LIN {X 0,Y 412.811,Z 882.496,A -85,B 0,C 180,E1 9709.918,E2 9709.918} C_VEL
LIN {X 0,Y 400.987,Z 919.927,A -85,B 0,C 180,E1 9708.865,E2 9708.865} C_VEL
LIN {X 0,Y 390.445,Z 950.291,A -85,B 0,C 180,E1 9707.777,E2 9707.777} C_VEL
LIN {X 0,Y 381.073,Z 973.005,A -85,B 0,C 180,E1 9706.758,E2 9706.758} C_VEL
LIN {X 0,Y 370.343,Z 995.885,A -85,B 0,C 180,E1 9705.507,E2 9705.507} C_VEL
LIN {X 0,Y 359.142,Z 1016.75,A -85,B 0,C 180,E1 9704.125,E2 9704.125} C_VEL
LIN {X 0,Y 346.722,Z 1037.419,A -85,B 0,C 180,E1 9702.455,E2 9702.455} C_VEL
LIN {X 0,Y 333.977,Z 1056.717,A -85,B 0,C 180,E1 9700.566,E2 9700.566} C_VEL
LIN {X 0,Y 320.046,Z 1075.683,A -85,B 0,C 180,E1 9698.278,E2 9698.278} C_VEL
LIN {X 0,Y 305.349,Z 1094.042,A -85,B 0,C 180,E1 9695.544,E2 9695.544} C_VEL
LIN {X 0,Y 291.757,Z 1109.715,A -85,B 0,C 180,E1 9692.662,E2 9692.662} C_VEL
LIN {X 0,Y 277.905,Z 1124.551,A -85,B 0,C 180,E1 9689.275,E2 9689.275} C_VEL
LIN {X 0,Y 264,Z 1138.62,A -85,B 0,C 180,E1 9685.267,E2 9685.267} C_VEL
LIN {X 0,Y 251.34,Z 1150.739,A -85,B 0,C 180,E1 9680.868,E2 9680.868} C_VEL
LIN {X 0,Y 239.156,Z 1162.034,A -85,B 0,C 180,E1 9675.633,E2 9675.633} C_VEL
LIN {X 0,Y 228.894,Z 1171.576,A -85,B 0,C 180,E1 9669.947,E2 9669.947} C_VEL
LIN {X 0,Y 220.104,Z 1179.984,A -85,B 0,C 180,E1 9663.341,E2 9663.341} C_VEL
LIN {X 0,Y 214.036,Z 1186.297,A -85,B 0,C 180,E1 9656.642,E2 9656.642} C_VEL
LIN {X 0,Y 210.026,Z 1191.417,A -85,B 0,C 180,E1 9649.174,E2 9649.174} C_VEL
LIN {X 0,Y 208.387,Z 1194.571,A -85,B 0,C 180,E1 9642.466,E2 9642.466} C_VEL
LIN {X 0,Y 208.029,Z 1196.144,A -85,B 0,C 180,E1 9636.621,E2 9636.621} C_VEL
LIN {X 0,Y 208.033,Z 1196.749,A -85,B 0,C 180,E1 9631.649,E2 9631.649} C_VEL
LIN {X 0,Y 208.017,Z 1196.626,A -85,B 0,C 180,E1 9626.414,E2 9626.414} C_VEL
LIN {X 0,Y 208.118,Z 1195.498,A -85,B 0,C 180,E1 9620.595,E2 9620.595} C_VEL
LIN {X 0,Y 209.018,Z 1193.143,A -85,B 0,C 180,E1 9614.173,E2 9614.173} C_VEL
LIN {X 0,Y 211.787,Z 1188.974,A -85,B 0,C 180,E1 9606.926,E2 9606.926} C_VEL
LIN {X 0,Y 216.9,Z 1183.182,A -85,B 0,C 180,E1 9599.832,E2 9599.832} C_VEL
LIN {X 0,Y 224.53,Z 1175.655,A -85,B 0,C 180,E1 9593.042,E2 9593.042} C_VEL
LIN {X 0,Y 234.651,Z 1166.193,A -85,B 0,C 180,E1 9586.679,E2 9586.679} C_VEL
LIN {X 0,Y 246.387,Z 1155.288,A -85,B 0,C 180,E1 9581.104,E2 9581.104} C_VEL
LIN {X 0,Y 259.941,Z 1142.471,A -85,B 0,C 180,E1 9576.053,E2 9576.053} C_VEL
LIN {X 0,Y 274.508,Z 1128.008,A -85,B 0,C 180,E1 9571.636,E2 9571.636} C_VEL
LIN {X 0,Y 289.503,Z 1112.12,A -85,B 0,C 180,E1 9567.846,E2 9567.846} C_VEL
LIN {X 0,Y 304.615,Z 1094.805,A -85,B 0,C 180,E1 9564.595,E2 9564.595} C_VEL
LIN {X 0,Y 319.981,Z 1075.607,A -85,B 0,C 180,E1 9561.727,E2 9561.727} C_VEL
LIN {X 0,Y 328.871,Z 1063.516,A -85,B 0,C 180,E1 9560.187,E2 9560.187} C_VEL
LIN {X 0,Y 312.273,Z 1075.955,A -85,B 0,C 180,E1 9558.869,E2 9558.869} C_VEL
LIN {X 0,Y 297.771,Z 1085.65,A -85,B 0,C 180,E1 9557.389,E2 9557.389} C_VEL
LIN {X 0,Y 282.8,Z 1094.747,A -85,B 0,C 180,E1 9555.483,E2 9555.483} C_VEL
LIN {X 0,Y 266.567,Z 1103.684,A -85,B 0,C 180,E1 9552.764,E2 9552.764} C_VEL
LIN {X 0,Y 252.428,Z 1110.885,A -85,B 0,C 180,E1 9549.577,E2 9549.577} C_VEL
LIN {X 0,Y 239.931,Z 1116.966,A -85,B 0,C 180,E1 9545.74,E2 9545.74} C_VEL
LIN {X 0,Y 229.73,Z 1121.893,A -85,B 0,C 180,E1 9541.247,E2 9541.247} C_VEL
LIN {X 0,Y 222.245,Z 1125.755,A -85,B 0,C 180,E1 9536.13,E2 9536.13} C_VEL
LIN {X 0,Y 217.444,Z 1129.147,A -85,B 0,C 180,E1 9529.936,E2 9529.936} C_VEL
LIN {X 0,Y 216.311,Z 1132.47,A -85,B 0,C 180,E1 9522.227,E2 9522.227} C_VEL
LIN {X 0,Y 222.255,Z 1135.612,A -85,B 0,C 180,E1 9512.394,E2 9512.394} C_VEL
LIN {X 0,Y 232.046,Z 1137.189,A -85,B 0,C 180,E1 9505.633,E2 9505.633} C_VEL
LIN {X 0,Y 243.185,Z 1137.819,A -85,B 0,C 180,E1 9500.714,E2 9500.714} C_VEL
LIN {X 0,Y 248.344,Z 1138.002,A -85,B 0,C 180,E1 9498.89,E2 9498.89} C_VEL
LIN {X 0,Y 235.847,Z 1150.144,A -85,B 0,C 180,E1 9493.048,E2 9493.048} C_VEL
LIN {X 0,Y 226.4,Z 1159.496,A -85,B 0,C 180,E1 9487.236,E2 9487.236} C_VEL
LIN {X 0,Y 218.613,Z 1167.518,A -85,B 0,C 180,E1 9480.697,E2 9480.697} C_VEL
LIN {X 0,Y 213.472,Z 1173.506,A -85,B 0,C 180,E1 9474.345,E2 9474.345} C_VEL
LIN {X 0,Y 210.092,Z 1178.183,A -85,B 0,C 180,E1 9467.451,E2 9467.451} C_VEL
LIN {X 0,Y 208.659,Z 1180.906,A -85,B 0,C 180,E1 9461.614,E2 9461.614} C_VEL
LIN {X 0,Y 208.156,Z 1182.441,A -85,B 0,C 180,E1 9456.346,E2 9456.346} C_VEL
LIN {X 0,Y 208.039,Z 1183.097,A -85,B 0,C 180,E1 9451.105,E2 9451.105} C_VEL
LIN {X 0,Y 208.082,Z 1182.855,A -85,B 0,C 180,E1 9445.594,E2 9445.594} C_VEL
LIN {X 0,Y 208.499,Z 1181.364,A -85,B 0,C 180,E1 9439.457,E2 9439.457} C_VEL
LIN {X 0,Y 209.703,Z 1178.846,A -85,B 0,C 180,E1 9433.665,E2 9433.665} C_VEL
LIN {X 0,Y 212.119,Z 1175.235,A -85,B 0,C 180,E1 9427.849,E2 9427.849} C_VEL
LIN {X 0,Y 217.157,Z 1169.21,A -85,B 0,C 180,E1 9420.79,E2 9420.79} C_VEL
LIN {X 0,Y 223.269,Z 1162.652,A -85,B 0,C 180,E1 9415.028,E2 9415.028} C_VEL
LIN {X 0,Y 232.367,Z 1153.659,A -85,B 0,C 180,E1 9408.829,E2 9408.829} C_VEL
LIN {X 0,Y 242.696,Z 1143.563,A -85,B 0,C 180,E1 9403.475,E2 9403.475} C_VEL
LIN {X 0,Y 255.719,Z 1130.948,A -85,B 0,C 180,E1 9398.199,E2 9398.199} C_VEL
LIN {X 0,Y 269.356,Z 1117.324,A -85,B 0,C 180,E1 9393.751,E2 9393.751} C_VEL
LIN {X 0,Y 283.658,Z 1102.296,A -85,B 0,C 180,E1 9389.878,E2 9389.878} C_VEL
LIN {X 0,Y 298.703,Z 1085.671,A -85,B 0,C 180,E1 9386.437,E2 9386.437} C_VEL
LIN {X 0,Y 313.12,Z 1068.459,A -85,B 0,C 180,E1 9383.591,E2 9383.591} C_VEL
LIN {X 0,Y 328.199,Z 1048.906,A -85,B 0,C 180,E1 9380.976,E2 9380.976} C_VEL
LIN {X 0,Y 341.827,Z 1029.717,A -85,B 0,C 180,E1 9378.875,E2 9378.875} C_VEL
LIN {X 0,Y 354.578,Z 1009.676,A -85,B 0,C 180,E1 9377.077,E2 9377.077} C_VEL
LIN {X 0,Y 366.366,Z 989.445,A -85,B 0,C 180,E1 9375.557,E2 9375.557} C_VEL
LIN {X 0,Y 377.497,Z 967.721,A -85,B 0,C 180,E1 9374.213,E2 9374.213} C_VEL
LIN {X 0,Y 388.399,Z 943.457,A -85,B 0,C 180,E1 9372.97,E2 9372.97} C_VEL
LIN {X 0,Y 397.147,Z 920.974,A -85,B 0,C 180,E1 9372.021,E2 9372.021} C_VEL
LIN {X 0,Y 404.369,Z 898.632,A -85,B 0,C 180,E1 9371.242,E2 9371.242} C_VEL
LIN {X 0,Y 414.435,Z 862.441,A -85,B 0,C 180,E1 9370.241,E2 9370.241} C_VEL
LIN {X 0,Y 426.056,Z 818.405,A -85,B 0,C 180,E1 9369.31,E2 9369.31} C_VEL
LIN {X 0,Y 438.723,Z 764.98,A -85,B 0,C 180,E1 9368.335,E2 9368.335} C_VEL
LIN {X 0,Y 449.507,Z 713.302,A -85,B 0,C 180,E1 9367.481,E2 9367.481} C_VEL
LIN {X 0,Y 450.16,Z 709.951,A -85,B 0,C 180,E1 9367.428,E2 9367.428} C_VEL
LIN {X 0,Y 450.433,Z 708.03,A -85,B 0,C 180,E1 9367.262,E2 9367.262} C_VEL
LIN {X 0,Y 450.405,Z 706.776,A -85,B 0,C 180,E1 9366.857,E2 9366.857} C_VEL
LIN {X 0,Y 449.978,Z 706.897,A -85,B 0,C 180,E1 9366.225,E2 9366.225} C_VEL
LIN {X 0,Y 449.184,Z 708.816,A -85,B 0,C 180,E1 9365.494,E2 9365.494} C_VEL
LIN {X 0,Y 447.901,Z 713.065,A -85,B 0,C 180,E1 9364.548,E2 9364.548} C_VEL
LIN {X 0,Y 446.794,Z 717.422,A -85,B 0,C 180,E1 9363.944,E2 9363.944} C_VEL
LIN {X 0,Y 446.052,Z 720.595,A -85,B 0,C 180,E1 9363.669,E2 9363.669} C_VEL
LIN {X 0,Y 439.226,Z 751.426,A -85,B 0,C 180,E1 9361.414,E2 9361.414} C_VEL
LIN {X 0,Y 433.442,Z 778.701,A -85,B 0,C 180,E1 9359.091,E2 9359.091} C_VEL
LIN {X 0,Y 428.161,Z 805.619,A -85,B 0,C 180,E1 9356.469,E2 9356.469} C_VEL
LIN {X 0,Y 423.543,Z 833.332,A -85,B 0,C 180,E1 9353.323,E2 9353.323} C_VEL
LIN {X 0,Y 421.82,Z 845.943,A -85,B 0,C 180,E1 9351.764,E2 9351.764} C_VEL
LIN {X 0,Y 410.531,Z 884.456,A -85,B 0,C 180,E1 9350.964,E2 9350.964} C_VEL
LIN {X 0,Y 399.026,Z 920.276,A -85,B 0,C 180,E1 9349.979,E2 9349.979} C_VEL
LIN {X 0,Y 389.372,Z 947.984,A -85,B 0,C 180,E1 9349.024,E2 9349.024} C_VEL
LIN {X 0,Y 380.15,Z 970.147,A -85,B 0,C 180,E1 9348.071,E2 9348.071} C_VEL
LIN {X 0,Y 370.437,Z 991.045,A -85,B 0,C 180,E1 9346.999,E2 9346.999} C_VEL
LIN {X 0,Y 358.755,Z 1012.769,A -85,B 0,C 180,E1 9345.638,E2 9345.638} C_VEL
LIN {X 0,Y 345.857,Z 1034.272,A -85,B 0,C 180,E1 9343.992,E2 9343.992} C_VEL
LIN {X 0,Y 333.329,Z 1053.021,A -85,B 0,C 180,E1 9342.242,E2 9342.242} C_VEL
LIN {X 0,Y 318.984,Z 1072.455,A -85,B 0,C 180,E1 9340.021,E2 9340.021} C_VEL
LIN {X 0,Y 305.01,Z 1089.89,A -85,B 0,C 180,E1 9337.579,E2 9337.579} C_VEL
LIN {X 0,Y 290.724,Z 1106.062,A -85,B 0,C 180,E1 9334.754,E2 9334.754} C_VEL
LIN {X 0,Y 275.774,Z 1121.883,A -85,B 0,C 180,E1 9331.327,E2 9331.327} C_VEL
LIN {X 0,Y 261.809,Z 1135.683,A -85,B 0,C 180,E1 9327.562,E2 9327.562} C_VEL
LIN {X 0,Y 248.369,Z 1148.138,A -85,B 0,C 180,E1 9323.233,E2 9323.233} C_VEL
LIN {X 0,Y 235.833,Z 1159.442,A -85,B 0,C 180,E1 9318.258,E2 9318.258} C_VEL
LIN {X 0,Y 224.154,Z 1169.717,A -85,B 0,C 180,E1 9312.338,E2 9312.338} C_VEL
LIN {X 0,Y 215.079,Z 1177.78,A -85,B 0,C 180,E1 9306.182,E2 9306.182} C_VEL
LIN {X 0,Y 207.746,Z 1184.836,A -85,B 0,C 180,E1 9299.081,E2 9299.081} C_VEL
LIN {X 0,Y 203.146,Z 1190.016,A -85,B 0,C 180,E1 9291.963,E2 9291.963} C_VEL
LIN {X 0,Y 200.806,Z 1193.468,A -85,B 0,C 180,E1 9284.982,E2 9284.982} C_VEL
LIN {X 0,Y 200.073,Z 1195.622,A -85,B 0,C 180,E1 9278.296,E2 9278.296} C_VEL
LIN {X 0,Y 200.028,Z 1196.434,A -85,B 0,C 180,E1 9272.575,E2 9272.575} C_VEL
LIN {X 0,Y 200.03,Z 1196.45,A -85,B 0,C 180,E1 9267.705,E2 9267.705} C_VEL
LIN {X 0,Y 200.058,Z 1195.716,A -85,B 0,C 180,E1 9262.241,E2 9262.241} C_VEL
LIN {X 0,Y 200.693,Z 1193.696,A -85,B 0,C 180,E1 9255.572,E2 9255.572} C_VEL
LIN {X 0,Y 202.881,Z 1190.321,A -85,B 0,C 180,E1 9248.607,E2 9248.607} C_VEL
LIN {X 0,Y 207.413,Z 1185.146,A -85,B 0,C 180,E1 9241.329,E2 9241.329} C_VEL
LIN {X 0,Y 214.755,Z 1178.072,A -85,B 0,C 180,E1 9234.077,E2 9234.077} C_VEL
LIN {X 0,Y 224.587,Z 1169.279,A -85,B 0,C 180,E1 9227.408,E2 9227.408} C_VEL
LIN {X 0,Y 236.348,Z 1158.936,A -85,B 0,C 180,E1 9221.509,E2 9221.509} C_VEL
LIN {X 0,Y 249.547,Z 1147.037,A -85,B 0,C 180,E1 9216.35,E2 9216.35} C_VEL
LIN {X 0,Y 264.395,Z 1133.053,A -85,B 0,C 180,E1 9211.686,E2 9211.686} C_VEL
LIN {X 0,Y 279.252,Z 1118.218,A -85,B 0,C 180,E1 9207.818,E2 9207.818} C_VEL
LIN {X 0,Y 294.414,Z 1101.886,A -85,B 0,C 180,E1 9204.466,E2 9204.466} C_VEL
LIN {X 0,Y 309.643,Z 1084.032,A -85,B 0,C 180,E1 9201.561,E2 9201.561} C_VEL
LIN {X 0,Y 315.577,Z 1076.646,A -85,B 0,C 180,E1 9200.52,E2 9200.52} C_VEL
LIN {X 0,Y 298.12,Z 1088.173,A -85,B 0,C 180,E1 9198.942,E2 9198.942} C_VEL
LIN {X 0,Y 281.163,Z 1098.148,A -85,B 0,C 180,E1 9196.929,E2 9196.929} C_VEL
LIN {X 0,Y 264.092,Z 1107.202,A -85,B 0,C 180,E1 9194.238,E2 9194.238} C_VEL
LIN {X 0,Y 250.119,Z 1113.928,A -85,B 0,C 180,E1 9191.296,E2 9191.296} C_VEL
LIN {X 0,Y 237.074,Z 1119.968,A -85,B 0,C 180,E1 9187.617,E2 9187.617} C_VEL
LIN {X 0,Y 227.218,Z 1124.381,A -85,B 0,C 180,E1 9183.785,E2 9183.785} C_VEL
LIN {X 0,Y 218.049,Z 1128.64,A -85,B 0,C 180,E1 9178.613,E2 9178.613} C_VEL
LIN {X 0,Y 211.262,Z 1132.587,A -85,B 0,C 180,E1 9171.563,E2 9171.563} C_VEL
LIN {X 0,Y 209.204,Z 1136.12,A -85,B 0,C 180,E1 9162.763,E2 9162.763} C_VEL
LIN {X 0,Y 215.054,Z 1139.294,A -85,B 0,C 180,E1 9152.293,E2 9152.293} C_VEL
LIN {X 0,Y 225.258,Z 1140.856,A -85,B 0,C 180,E1 9145.067,E2 9145.067} C_VEL
LIN {X 0,Y 237.163,Z 1141.564,A -85,B 0,C 180,E1 9139.83,E2 9139.83} C_VEL
LIN {X 0,Y 239.46,Z 1141.692,A -85,B 0,C 180,E1 9138.933,E2 9138.933} C_VEL
LIN {X 0,Y 228.015,Z 1152.144,A -85,B 0,C 180,E1 9133.513,E2 9133.513} C_VEL
LIN {X 0,Y 218.012,Z 1161.542,A -85,B 0,C 180,E1 9127.261,E2 9127.261} C_VEL
LIN {X 0,Y 210.559,Z 1168.836,A -85,B 0,C 180,E1 9120.858,E2 9120.858} C_VEL
LIN {X 0,Y 204.789,Z 1175.208,A -85,B 0,C 180,E1 9113.376,E2 9113.376} C_VEL
LIN {X 0,Y 201.976,Z 1178.973,A -85,B 0,C 180,E1 9107.164,E2 9107.164} C_VEL
LIN {X 0,Y 200.563,Z 1181.603,A -85,B 0,C 180,E1 9100.924,E2 9100.924} C_VEL
LIN {X 0,Y 200.092,Z 1183.11,A -85,B 0,C 180,E1 9094.589,E2 9094.589} C_VEL
LIN {X 0,Y 200.043,Z 1183.37,A -85,B 0,C 180,E1 9088.858,E2 9088.858} C_VEL
LIN {X 0,Y 200.17,Z 1182.736,A -85,B 0,C 180,E1 9083.406,E2 9083.406} C_VEL
LIN {X 0,Y 200.718,Z 1181.223,A -85,B 0,C 180,E1 9077.927,E2 9077.927} C_VEL
LIN {X 0,Y 202.181,Z 1178.677,A -85,B 0,C 180,E1 9072.148,E2 9072.148} C_VEL
LIN {X 0,Y 205.577,Z 1174.375,A -85,B 0,C 180,E1 9065.278,E2 9065.278} C_VEL
LIN {X 0,Y 211.111,Z 1168.293,A -85,B 0,C 180,E1 9058.489,E2 9058.489} C_VEL
LIN {X 0,Y 218.999,Z 1160.714,A -85,B 0,C 180,E1 9051.953,E2 9051.953} C_VEL
LIN {X 0,Y 228.792,Z 1151.499,A -85,B 0,C 180,E1 9045.988,E2 9045.988} C_VEL
LIN {X 0,Y 240.607,Z 1140.727,A -85,B 0,C 180,E1 9040.498,E2 9040.498} C_VEL
LIN {X 0,Y 254.213,Z 1127.965,A -85,B 0,C 180,E1 9035.499,E2 9035.499} C_VEL
LIN {X 0,Y 269.411,Z 1113.153,A -85,B 0,C 180,E1 9030.988,E2 9030.988} C_VEL
LIN {X 0,Y 284.568,Z 1097.649,A -85,B 0,C 180,E1 9027.263,E2 9027.263} C_VEL
LIN {X 0,Y 300.298,Z 1080.229,A -85,B 0,C 180,E1 9023.968,E2 9023.968} C_VEL
LIN {X 0,Y 316.161,Z 1061.208,A -85,B 0,C 180,E1 9021.106,E2 9021.106} C_VEL
LIN {X 0,Y 330.628,Z 1042.445,A -85,B 0,C 180,E1 9018.822,E2 9018.822} C_VEL
LIN {X 0,Y 344.691,Z 1022.113,A -85,B 0,C 180,E1 9016.819,E2 9016.819} C_VEL
LIN {X 0,Y 358.519,Z 999.958,A -85,B 0,C 180,E1 9015.033,E2 9015.033} C_VEL
LIN {X 0,Y 370.366,Z 978.771,A -85,B 0,C 180,E1 9013.625,E2 9013.625} C_VEL
LIN {X 0,Y 380.429,Z 958.054,A -85,B 0,C 180,E1 9012.479,E2 9012.479} C_VEL
LIN {X 0,Y 389.747,Z 936.743,A -85,B 0,C 180,E1 9011.487,E2 9011.487} C_VEL
LIN {X 0,Y 397.779,Z 914.776,A -85,B 0,C 180,E1 9010.641,E2 9010.641} C_VEL
LIN {X 0,Y 404.743,Z 893.101,A -85,B 0,C 180,E1 9009.944,E2 9009.944} C_VEL
LIN {X 0,Y 416.476,Z 850.737,A -85,B 0,C 180,E1 9008.867,E2 9008.867} C_VEL
LIN {X 0,Y 429.491,Z 800.675,A -85,B 0,C 180,E1 9007.911,E2 9007.911} C_VEL
LIN {X 0,Y 441.609,Z 748.272,A -85,B 0,C 180,E1 9007.011,E2 9007.011} C_VEL
LIN {X 0,Y 452.336,Z 694.609,A -85,B 0,C 180,E1 9006.178,E2 9006.178} C_VEL
LIN {X 0,Y 452.794,Z 692.087,A -85,B 0,C 180,E1 9006.121,E2 9006.121} C_VEL
LIN {X 0,Y 452.304,Z 692.999,A -85,B 0,C 180,E1 9005.574,E2 9005.574} C_VEL
LIN {X 0,Y 446.052,Z 720.595,A -85,B 0,C 180,E1 9003.669,E2 9003.669} C_VEL
LIN {X 0,Y 444.49,Z 727.708,A -85,B 0,C 180,E1 9003.32,E2 9003.32} C_VEL
LIN {X 0,Y 440.022,Z 747.992,A -85,B 0,C 180,E1 9002.766,E2 9002.766} C_VEL
LIN {X 0,Y 438.677,Z 753.942,A -85,B 0,C 180,E1 9002.427,E2 9002.427} C_VEL
LIN {X 0,Y 432.402,Z 781.506,A -85,B 0,C 180,E1 9000.099,E2 9000.099} C_VEL
LIN {X 0,Y 426.937,Z 806.918,A -85,B 0,C 180,E1 8997.651,E2 8997.651} C_VEL
LIN {X 0,Y 421.776,Z 834.64,A -85,B 0,C 180,E1 8994.559,E2 8994.559} C_VEL
LIN {X 0,Y 419.509,Z 849.049,A -85,B 0,C 180,E1 8992.782,E2 8992.782} C_VEL
LIN {X 0,Y 407.591,Z 888.947,A -85,B 0,C 180,E1 8991.962,E2 8991.962} C_VEL
LIN {X 0,Y 395.608,Z 925.572,A -85,B 0,C 180,E1 8990.955,E2 8990.955} C_VEL
LIN {X 0,Y 386.691,Z 950.05,A -85,B 0,C 180,E1 8990.106,E2 8990.106} C_VEL
LIN {X 0,Y 378.853,Z 968.601,A -85,B 0,C 180,E1 8989.329,E2 8989.329} C_VEL
LIN {X 0,Y 369.103,Z 989.382,A -85,B 0,C 180,E1 8988.306,E2 8988.306} C_VEL
LIN {X 0,Y 358.011,Z 1009.79,A -85,B 0,C 180,E1 8987.077,E2 8987.077} C_VEL
LIN {X 0,Y 346.237,Z 1029.583,A -85,B 0,C 180,E1 8985.657,E2 8985.657} C_VEL
LIN {X 0,Y 332.966,Z 1049.316,A -85,B 0,C 180,E1 8983.925,E2 8983.925} C_VEL
LIN {X 0,Y 317.96,Z 1069.51,A -85,B 0,C 180,E1 8981.74,E2 8981.74} C_VEL
LIN {X 0,Y 304.238,Z 1086.387,A -85,B 0,C 180,E1 8979.489,E2 8979.489} C_VEL
LIN {X 0,Y 288.712,Z 1103.847,A -85,B 0,C 180,E1 8976.594,E2 8976.594} C_VEL
LIN {X 0,Y 273.228,Z 1119.915,A -85,B 0,C 180,E1 8973.236,E2 8973.236} C_VEL
LIN {X 0,Y 259.02,Z 1133.559,A -85,B 0,C 180,E1 8969.622,E2 8969.622} C_VEL
LIN {X 0,Y 244.002,Z 1147.15,A -85,B 0,C 180,E1 8965.036,E2 8965.036} C_VEL
LIN {X 0,Y 230.815,Z 1158.549,A -85,B 0,C 180,E1 8960.058,E2 8960.058} C_VEL
LIN {X 0,Y 218.904,Z 1168.528,A -85,B 0,C 180,E1 8954.33,E2 8954.33} C_VEL
LIN {X 0,Y 208.625,Z 1177.205,A -85,B 0,C 180,E1 8947.739,E2 8947.739} C_VEL
LIN {X 0,Y 200.7,Z 1184.31,A -85,B 0,C 180,E1 8940.47,E2 8940.47} C_VEL
LIN {X 0,Y 195.6,Z 1189.596,A -85,B 0,C 180,E1 8933.052,E2 8933.052} C_VEL
LIN {X 0,Y 192.933,Z 1193.182,A -85,B 0,C 180,E1 8925.63,E2 8925.63} C_VEL
LIN {X 0,Y 192.08,Z 1195.378,A -85,B 0,C 180,E1 8918.48,E2 8918.48} C_VEL
LIN {X 0,Y 192.032,Z 1196.169,A -85,B 0,C 180,E1 8912.682,E2 8912.682} C_VEL
LIN {X 0,Y 192.033,Z 1196.186,A -85,B 0,C 180,E1 8907.609,E2 8907.609} C_VEL
LIN {X 0,Y 192.069,Z 1195.445,A -85,B 0,C 180,E1 8901.916,E2 8901.916} C_VEL
LIN {X 0,Y 192.801,Z 1193.412,A -85,B 0,C 180,E1 8894.968,E2 8894.968} C_VEL
LIN {X 0,Y 195.221,Z 1190.016,A -85,B 0,C 180,E1 8887.724,E2 8887.724} C_VEL
LIN {X 0,Y 200.259,Z 1184.711,A -85,B 0,C 180,E1 8880.043,E2 8880.043} C_VEL
LIN {X 0,Y 208.374,Z 1177.393,A -85,B 0,C 180,E1 8872.449,E2 8872.449} C_VEL
LIN {X 0,Y 218.914,Z 1168.479,A -85,B 0,C 180,E1 8865.663,E2 8865.663} C_VEL
LIN {X 0,Y 231.361,Z 1158.036,A -85,B 0,C 180,E1 8859.707,E2 8859.707} C_VEL
LIN {X 0,Y 245.377,Z 1145.87,A -85,B 0,C 180,E1 8854.501,E2 8854.501} C_VEL
LIN {X 0,Y 260.73,Z 1131.884,A -85,B 0,C 180,E1 8849.904,E2 8849.904} C_VEL
LIN {X 0,Y 276.89,Z 1116.111,A -85,B 0,C 180,E1 8845.91,E2 8845.91} C_VEL
LIN {X 0,Y 292.537,Z 1099.608,A -85,B 0,C 180,E1 8842.648,E2 8842.648} C_VEL
LIN {X 0,Y 302.365,Z 1088.426,A -85,B 0,C 180,E1 8840.806,E2 8840.806} C_VEL
LIN {X 0,Y 284.426,Z 1098.878,A -85,B 0,C 180,E1 8838.97,E2 8838.97} C_VEL
LIN {X 0,Y 267.69,Z 1107.72,A -85,B 0,C 180,E1 8836.715,E2 8836.715} C_VEL
LIN {X 0,Y 252.346,Z 1115.038,A -85,B 0,C 180,E1 8833.987,E2 8833.987} C_VEL
LIN {X 0,Y 238.031,Z 1121.349,A -85,B 0,C 180,E1 8830.582,E2 8830.582} C_VEL
LIN {X 0,Y 225.412,Z 1126.726,A -85,B 0,C 180,E1 8826.453,E2 8826.453} C_VEL
LIN {X 0,Y 215.059,Z 1131.104,A -85,B 0,C 180,E1 8821.504,E2 8821.504} C_VEL
LIN {X 0,Y 207.526,Z 1134.572,A -85,B 0,C 180,E1 8815.855,E2 8815.855} C_VEL
LIN {X 0,Y 202.41,Z 1138.234,A -85,B 0,C 180,E1 8807.446,E2 8807.446} C_VEL
LIN {X 0,Y 203.621,Z 1141.241,A -85,B 0,C 180,E1 8798.087,E2 8798.087} C_VEL
LIN {X 0,Y 210.765,Z 1143.45,A -85,B 0,C 180,E1 8789.495,E2 8789.495} C_VEL
LIN {X 0,Y 222.632,Z 1144.699,A -85,B 0,C 180,E1 8782.352,E2 8782.352} C_VEL
LIN {X 0,Y 230.538,Z 1145.066,A -85,B 0,C 180,E1 8779.001,E2 8779.001} C_VEL
LIN {X 0,Y 218.868,Z 1155.373,A -85,B 0,C 180,E1 8773.26,E2 8773.26} C_VEL
LIN {X 0,Y 208.902,Z 1164.124,A -85,B 0,C 180,E1 8766.752,E2 8766.752} C_VEL
LIN {X 0,Y 201.1,Z 1171.519,A -85,B 0,C 180,E1 8759.491,E2 8759.491} C_VEL
LIN {X 0,Y 196.371,Z 1176.499,A -85,B 0,C 180,E1 8752.77,E2 8752.77} C_VEL
LIN {X 0,Y 193.569,Z 1180.224,A -85,B 0,C 180,E1 8745.892,E2 8745.892} C_VEL
LIN {X 0,Y 192.354,Z 1182.536,A -85,B 0,C 180,E1 8738.975,E2 8738.975} C_VEL
LIN {X 0,Y 192.066,Z 1183.477,A -85,B 0,C 180,E1 8733.286,E2 8733.286} C_VEL
LIN {X 0,Y 192.05,Z 1183.589,A -85,B 0,C 180,E1 8728.214,E2 8728.214} C_VEL
LIN {X 0,Y 192.206,Z 1182.937,A -85,B 0,C 180,E1 8722.832,E2 8722.832} C_VEL
LIN {X 0,Y 192.852,Z 1181.391,A -85,B 0,C 180,E1 8717.122,E2 8717.122} C_VEL
LIN {X 0,Y 194.65,Z 1178.667,A -85,B 0,C 180,E1 8710.811,E2 8710.811} C_VEL
LIN {X 0,Y 198.945,Z 1173.722,A -85,B 0,C 180,E1 8703.111,E2 8703.111} C_VEL
LIN {X 0,Y 204.582,Z 1168.146,A -85,B 0,C 180,E1 8696.816,E2 8696.816} C_VEL
LIN {X 0,Y 213.277,Z 1160.304,A -85,B 0,C 180,E1 8690.043,E2 8690.043} C_VEL
LIN {X 0,Y 223.85,Z 1151.036,A -85,B 0,C 180,E1 8684.021,E2 8684.021} C_VEL
LIN {X 0,Y 237.519,Z 1139.058,A -85,B 0,C 180,E1 8678.08,E2 8678.08} C_VEL
LIN {X 0,Y 252.012,Z 1126.11,A -85,B 0,C 180,E1 8673.164,E2 8673.164} C_VEL
LIN {X 0,Y 267.301,Z 1111.6,A -85,B 0,C 180,E1 8668.924,E2 8668.924} C_VEL
LIN {X 0,Y 283.809,Z 1094.958,A -85,B 0,C 180,E1 8665.125,E2 8665.125} C_VEL
LIN {X 0,Y 299.806,Z 1077.677,A -85,B 0,C 180,E1 8662.012,E2 8662.012} C_VEL
LIN {X 0,Y 314.919,Z 1059.732,A -85,B 0,C 180,E1 8659.448,E2 8659.448} C_VEL
LIN {X 0,Y 330.581,Z 1039.479,A -85,B 0,C 180,E1 8657.111,E2 8657.111} C_VEL
LIN {X 0,Y 344.997,Z 1018.928,A -85,B 0,C 180,E1 8655.189,E2 8655.189} C_VEL
LIN {X 0,Y 357.103,Z 999.454,A -85,B 0,C 180,E1 8653.7,E2 8653.7} C_VEL
LIN {X 0,Y 368.546,Z 979.309,A -85,B 0,C 180,E1 8652.404,E2 8652.404} C_VEL
LIN {X 0,Y 378.32,Z 959.508,A -85,B 0,C 180,E1 8651.335,E2 8651.335} C_VEL
LIN {X 0,Y 387.728,Z 938.49,A -85,B 0,C 180,E1 8650.375,E2 8650.375} C_VEL
LIN {X 0,Y 395.921,Z 916.579,A -85,B 0,C 180,E1 8649.546,E2 8649.546} C_VEL
LIN {X 0,Y 403.228,Z 894.205,A -85,B 0,C 180,E1 8648.841,E2 8648.841} C_VEL
LIN {X 0,Y 415.5,Z 850.931,A -85,B 0,C 180,E1 8647.769,E2 8647.769} C_VEL
LIN {X 0,Y 429.41,Z 798.024,A -85,B 0,C 180,E1 8646.796,E2 8646.796} C_VEL
LIN {X 0,Y 442.417,Z 741.668,A -85,B 0,C 180,E1 8645.867,E2 8645.867} C_VEL
LIN {X 0,Y 448.433,Z 712.167,A -85,B 0,C 180,E1 8645.401,E2 8645.401} C_VEL
LIN {X 0,Y 439.649,Z 749.613,A -85,B 0,C 180,E1 8642.754,E2 8642.754} C_VEL
LIN {X 0,Y 438.677,Z 753.942,A -85,B 0,C 180,E1 8642.427,E2 8642.427} C_VEL
LIN {X 0,Y 437.092,Z 760.897,A -85,B 0,C 180,E1 8642.026,E2 8642.026} C_VEL
LIN {X 0,Y 432.325,Z 780.783,A -85,B 0,C 180,E1 8641.3,E2 8641.3} C_VEL
LIN {X 0,Y 430.941,Z 786.563,A -85,B 0,C 180,E1 8640.91,E2 8640.91} C_VEL
LIN {X 0,Y 425.125,Z 812.174,A -85,B 0,C 180,E1 8638.435,E2 8638.435} C_VEL
LIN {X 0,Y 419.318,Z 841.092,A -85,B 0,C 180,E1 8635.178,E2 8635.178} C_VEL
LIN {X 0,Y 417.366,Z 852.094,A -85,B 0,C 180,E1 8633.813,E2 8633.813} C_VEL
LIN {X 0,Y 405.206,Z 892.313,A -85,B 0,C 180,E1 8633.002,E2 8633.002} C_VEL
LIN {X 0,Y 392.778,Z 929.723,A -85,B 0,C 180,E1 8631.982,E2 8631.982} C_VEL
LIN {X 0,Y 384.439,Z 951.566,A -85,B 0,C 180,E1 8631.226,E2 8631.226} C_VEL
LIN {X 0,Y 374.842,Z 973.68,A -85,B 0,C 180,E1 8630.307,E2 8630.307} C_VEL
LIN {X 0,Y 364.785,Z 993.544,A -85,B 0,C 180,E1 8629.3,E2 8629.3} C_VEL
LIN {X 0,Y 353.562,Z 1013.799,A -85,B 0,C 180,E1 8628.085,E2 8628.085} C_VEL
LIN {X 0,Y 340.805,Z 1033.918,A -85,B 0,C 180,E1 8626.598,E2 8626.598} C_VEL
LIN {X 0,Y 327.732,Z 1052.851,A -85,B 0,C 180,E1 8624.921,E2 8624.921} C_VEL
LIN {X 0,Y 312.912,Z 1071.98,A -85,B 0,C 180,E1 8622.82,E2 8622.82} C_VEL
LIN {X 0,Y 297.337,Z 1090.303,A -85,B 0,C 180,E1 8620.311,E2 8620.311} C_VEL
LIN {X 0,Y 282.353,Z 1106.507,A -85,B 0,C 180,E1 8617.55,E2 8617.55} C_VEL
LIN {X 0,Y 266.576,Z 1122.14,A -85,B 0,C 180,E1 8614.177,E2 8614.177} C_VEL
LIN {X 0,Y 251.062,Z 1136.44,A -85,B 0,C 180,E1 8610.245,E2 8610.245} C_VEL
LIN {X 0,Y 237.359,Z 1148.247,A -85,B 0,C 180,E1 8606.079,E2 8606.079} C_VEL
LIN {X 0,Y 223.251,Z 1159.861,A -85,B 0,C 180,E1 8600.783,E2 8600.783} C_VEL
LIN {X 0,Y 211.06,Z 1169.665,A -85,B 0,C 180,E1 8594.895,E2 8594.895} C_VEL
LIN {X 0,Y 200.659,Z 1177.991,A -85,B 0,C 180,E1 8588.157,E2 8588.157} C_VEL
LIN {X 0,Y 192.811,Z 1184.627,A -85,B 0,C 180,E1 8580.886,E2 8580.886} C_VEL
LIN {X 0,Y 187.596,Z 1189.728,A -85,B 0,C 180,E1 8573.225,E2 8573.225} C_VEL
LIN {X 0,Y 184.949,Z 1193.1,A -85,B 0,C 180,E1 8565.777,E2 8565.777} C_VEL
LIN {X 0,Y 184.082,Z 1195.18,A -85,B 0,C 180,E1 8558.429,E2 8558.429} C_VEL
LIN {X 0,Y 184.035,Z 1195.906,A -85,B 0,C 180,E1 8552.799,E2 8552.799} C_VEL
LIN {X 0,Y 184.039,Z 1195.939,A -85,B 0,C 180,E1 8547.817,E2 8547.817} C_VEL
LIN {X 0,Y 184.065,Z 1195.279,A -85,B 0,C 180,E1 8542.191,E2 8542.191} C_VEL
LIN {X 0,Y 184.729,Z 1193.492,A -85,B 0,C 180,E1 8535.258,E2 8535.258} C_VEL
LIN {X 0,Y 187.151,Z 1190.191,A -85,B 0,C 180,E1 8527.704,E2 8527.704} C_VEL
LIN {X 0,Y 192.364,Z 1185.017,A -85,B 0,C 180,E1 8519.639,E2 8519.639} C_VEL
LIN {X 0,Y 200.423,Z 1178.158,A -85,B 0,C 180,E1 8512.022,E2 8512.022} C_VEL
LIN {X 0,Y 211.069,Z 1169.606,A -85,B 0,C 180,E1 8505.098,E2 8505.098} C_VEL
LIN {X 0,Y 223.808,Z 1159.349,A -85,B 0,C 180,E1 8498.976,E2 8498.976} C_VEL
LIN {X 0,Y 238.625,Z 1147.12,A -85,B 0,C 180,E1 8493.5,E2 8493.5} C_VEL
LIN {X 0,Y 254.497,Z 1133.28,A -85,B 0,C 180,E1 8488.815,E2 8488.815} C_VEL
LIN {X 0,Y 270.995,Z 1117.809,A -85,B 0,C 180,E1 8484.811,E2 8484.811} C_VEL
LIN {X 0,Y 287.018,Z 1101.46,A -85,B 0,C 180,E1 8481.537,E2 8481.537} C_VEL
LIN {X 0,Y 289.307,Z 1098.949,A -85,B 0,C 180,E1 8481.062,E2 8481.062} C_VEL
LIN {X 0,Y 271.912,Z 1108.059,A -85,B 0,C 180,E1 8479.076,E2 8479.076} C_VEL
LIN {X 0,Y 254.352,Z 1116.406,A -85,B 0,C 180,E1 8476.417,E2 8476.417} C_VEL
LIN {X 0,Y 238.16,Z 1123.312,A -85,B 0,C 180,E1 8473.078,E2 8473.078} C_VEL
LIN {X 0,Y 223.699,Z 1129.125,A -85,B 0,C 180,E1 8468.935,E2 8468.935} C_VEL
LIN {X 0,Y 211.883,Z 1133.733,A -85,B 0,C 180,E1 8464.059,E2 8464.059} C_VEL
LIN {X 0,Y 202.893,Z 1137.441,A -85,B 0,C 180,E1 8458.306,E2 8458.306} C_VEL
LIN {X 0,Y 196.877,Z 1140.612,A -85,B 0,C 180,E1 8451.236,E2 8451.236} C_VEL
LIN {X 0,Y 195.049,Z 1143.6,A -85,B 0,C 180,E1 8442.395,E2 8442.395} C_VEL
LIN {X 0,Y 201.304,Z 1146.465,A -85,B 0,C 180,E1 8431.196,E2 8431.196} C_VEL
LIN {X 0,Y 212.531,Z 1147.861,A -85,B 0,C 180,E1 8423.309,E2 8423.309} C_VEL
LIN {X 0,Y 221.655,Z 1148.402,A -85,B 0,C 180,E1 8419.101,E2 8419.101} C_VEL
LIN {X 0,Y 210.122,Z 1157.898,A -85,B 0,C 180,E1 8413.258,E2 8413.258} C_VEL
LIN {X 0,Y 201.204,Z 1165.4,A -85,B 0,C 180,E1 8407.325,E2 8407.325} C_VEL
LIN {X 0,Y 193.155,Z 1172.526,A -85,B 0,C 180,E1 8399.803,E2 8399.803} C_VEL
LIN {X 0,Y 188.482,Z 1177.17,A -85,B 0,C 180,E1 8393.118,E2 8393.118} C_VEL
LIN {X 0,Y 185.403,Z 1180.995,A -85,B 0,C 180,E1 8385.327,E2 8385.327} C_VEL
LIN {X 0,Y 184.333,Z 1182.927,A -85,B 0,C 180,E1 8378.74,E2 8378.74} C_VEL
LIN {X 0,Y 184.067,Z 1183.76,A -85,B 0,C 180,E1 8373.118,E2 8373.118} C_VEL
LIN {X 0,Y 184.054,Z 1183.854,A -85,B 0,C 180,E1 8368.136,E2 8368.136} C_VEL
LIN {X 0,Y 184.229,Z 1183.205,A -85,B 0,C 180,E1 8362.519,E2 8362.519} C_VEL
LIN {X 0,Y 184.953,Z 1181.663,A -85,B 0,C 180,E1 8356.562,E2 8356.562} C_VEL
LIN {X 0,Y 186.947,Z 1178.946,A -85,B 0,C 180,E1 8349.987,E2 8349.987} C_VEL
LIN {X 0,Y 191.623,Z 1174.011,A -85,B 0,C 180,E1 8341.995,E2 8341.995} C_VEL
LIN {X 0,Y 197.701,Z 1168.467,A -85,B 0,C 180,E1 8335.502,E2 8335.502} C_VEL
LIN {X 0,Y 207.387,Z 1160.276,A -85,B 0,C 180,E1 8328.296,E2 8328.296} C_VEL
LIN {X 0,Y 218.646,Z 1150.99,A -85,B 0,C 180,E1 8322.203,E2 8322.203} C_VEL
LIN {X 0,Y 232.794,Z 1139.167,A -85,B 0,C 180,E1 8316.352,E2 8316.352} C_VEL
LIN {X 0,Y 247.557,Z 1126.51,A -85,B 0,C 180,E1 8311.551,E2 8311.551} C_VEL
LIN {X 0,Y 263.388,Z 1112.031,A -85,B 0,C 180,E1 8307.344,E2 8307.344} C_VEL
LIN {X 0,Y 279.636,Z 1096.183,A -85,B 0,C 180,E1 8303.749,E2 8303.749} C_VEL
LIN {X 0,Y 296.022,Z 1079.061,A -85,B 0,C 180,E1 8300.678,E2 8300.678} C_VEL
LIN {X 0,Y 311.608,Z 1061.086,A -85,B 0,C 180,E1 8298.135,E2 8298.135} C_VEL
LIN {X 0,Y 327.42,Z 1041.16,A -85,B 0,C 180,E1 8295.865,E2 8295.865} C_VEL
LIN {X 0,Y 341.392,Z 1021.784,A -85,B 0,C 180,E1 8294.069,E2 8294.069} C_VEL
LIN {X 0,Y 353.502,Z 1002.924,A -85,B 0,C 180,E1 8292.633,E2 8292.633} C_VEL
LIN {X 0,Y 364.196,Z 984.701,A -85,B 0,C 180,E1 8291.454,E2 8291.454} C_VEL
LIN {X 0,Y 375.006,Z 963.873,A -85,B 0,C 180,E1 8290.318,E2 8290.318} C_VEL
LIN {X 0,Y 383.785,Z 944.873,A -85,B 0,C 180,E1 8289.447,E2 8289.447} C_VEL
LIN {X 0,Y 392.828,Z 922.225,A -85,B 0,C 180,E1 8288.573,E2 8288.573} C_VEL
LIN {X 0,Y 399.923,Z 901.452,A -85,B 0,C 180,E1 8287.904,E2 8287.904} C_VEL
LIN {X 0,Y 411.996,Z 860.655,A -85,B 0,C 180,E1 8286.868,E2 8286.868} C_VEL
LIN {X 0,Y 426.144,Z 808.526,A -85,B 0,C 180,E1 8285.902,E2 8285.902} C_VEL
LIN {X 0,Y 438.788,Z 755.89,A -85,B 0,C 180,E1 8285.044,E2 8285.044} C_VEL
LIN {X 0,Y 442.588,Z 738.476,A -85,B 0,C 180,E1 8284.762,E2 8284.762} C_VEL
LIN {X 0,Y 435.441,Z 767.749,A -85,B 0,C 180,E1 8282.533,E2 8282.533} C_VEL
LIN {X 0,Y 430.941,Z 786.563,A -85,B 0,C 180,E1 8280.91,E2 8280.91} C_VEL
LIN {X 0,Y 429.349,Z 793.362,A -85,B 0,C 180,E1 8280.452,E2 8280.452} C_VEL
LIN {X 0,Y 424.718,Z 811.92,A -85,B 0,C 180,E1 8279.623,E2 8279.623} C_VEL
LIN {X 0,Y 423.084,Z 818.472,A -85,B 0,C 180,E1 8279.114,E2 8279.114} C_VEL
LIN {X 0,Y 417.01,Z 846.356,A -85,B 0,C 180,E1 8275.944,E2 8275.944} C_VEL
LIN {X 0,Y 415.317,Z 855.237,A -85,B 0,C 180,E1 8274.852,E2 8274.852} C_VEL
LIN {X 0,Y 403.575,Z 893.556,A -85,B 0,C 180,E1 8274.099,E2 8274.099} C_VEL
LIN {X 0,Y 391.286,Z 930.132,A -85,B 0,C 180,E1 8273.133,E2 8273.133} C_VEL
LIN {X 0,Y 382.338,Z 953.222,A -85,B 0,C 180,E1 8272.355,E2 8272.355} C_VEL
LIN {X 0,Y 372.098,Z 975.729,A -85,B 0,C 180,E1 8271.428,E2 8271.428} C_VEL
LIN {X 0,Y 361.505,Z 996.346,A -85,B 0,C 180,E1 8270.4,E2 8270.4} C_VEL
LIN {X 0,Y 349.886,Z 1016.222,A -85,B 0,C 180,E1 8269.201,E2 8269.201} C_VEL
LIN {X 0,Y 339.337,Z 1032.592,A -85,B 0,C 180,E1 8268.02,E2 8268.02} C_VEL
LIN {X 0,Y 326.517,Z 1050.967,A -85,B 0,C 180,E1 8266.464,E2 8266.464} C_VEL
LIN {X 0,Y 312.222,Z 1069.167,A -85,B 0,C 180,E1 8264.557,E2 8264.557} C_VEL
LIN {X 0,Y 297.069,Z 1086.994,A -85,B 0,C 180,E1 8262.266,E2 8262.266} C_VEL
LIN {X 0,Y 281.602,Z 1103.446,A -85,B 0,C 180,E1 8259.608,E2 8259.608} C_VEL
LIN {X 0,Y 265.246,Z 1119.449,A -85,B 0,C 180,E1 8256.344,E2 8256.344} C_VEL
LIN {X 0,Y 249.79,Z 1133.506,A -85,B 0,C 180,E1 8252.696,E2 8252.696} C_VEL
LIN {X 0,Y 234.493,Z 1146.334,A -85,B 0,C 180,E1 8248.367,E2 8248.367} C_VEL
LIN {X 0,Y 219.744,Z 1158.089,A -85,B 0,C 180,E1 8243.204,E2 8243.204} C_VEL
LIN {X 0,Y 206.672,Z 1168.146,A -85,B 0,C 180,E1 8237.334,E2 8237.334} C_VEL
LIN {X 0,Y 195.319,Z 1176.692,A -85,B 0,C 180,E1 8230.547,E2 8230.547} C_VEL
LIN {X 0,Y 185.989,Z 1184.063,A -85,B 0,C 180,E1 8222.516,E2 8222.516} C_VEL
LIN {X 0,Y 180.127,Z 1189.331,A -85,B 0,C 180,E1 8214.443,E2 8214.443} C_VEL
LIN {X 0,Y 177.153,Z 1192.734,A -85,B 0,C 180,E1 8206.725,E2 8206.725} C_VEL
LIN {X 0,Y 176.1,Z 1194.895,A -85,B 0,C 180,E1 8198.896,E2 8198.896} C_VEL
LIN {X 0,Y 176.037,Z 1195.641,A -85,B 0,C 180,E1 8192.926,E2 8192.926} C_VEL
LIN {X 0,Y 176.042,Z 1195.676,A -85,B 0,C 180,E1 8187.717,E2 8187.717} C_VEL
LIN {X 0,Y 176.076,Z 1195.013,A -85,B 0,C 180,E1 8181.834,E2 8181.834} C_VEL
LIN {X 0,Y 176.921,Z 1193.091,A -85,B 0,C 180,E1 8174.256,E2 8174.256} C_VEL
LIN {X 0,Y 179.7,Z 1189.721,A -85,B 0,C 180,E1 8166.379,E2 8166.379} C_VEL
LIN {X 0,Y 185.43,Z 1184.505,A -85,B 0,C 180,E1 8158.096,E2 8158.096} C_VEL
LIN {X 0,Y 194.137,Z 1177.599,A -85,B 0,C 180,E1 8150.305,E2 8150.305} C_VEL
LIN {X 0,Y 205.683,Z 1168.841,A -85,B 0,C 180,E1 8143.177,E2 8143.177} C_VEL
LIN {X 0,Y 219.168,Z 1158.48,A -85,B 0,C 180,E1 8137.019,E2 8137.019} C_VEL
LIN {X 0,Y 234.708,Z 1146.101,A -85,B 0,C 180,E1 8131.563,E2 8131.563} C_VEL
LIN {X 0,Y 250.83,Z 1132.452,A -85,B 0,C 180,E1 8127.029,E2 8127.029} C_VEL
LIN {X 0,Y 266.778,Z 1117.932,A -85,B 0,C 180,E1 8123.322,E2 8123.322} C_VEL
LIN {X 0,Y 276.565,Z 1108.372,A -85,B 0,C 180,E1 8121.306,E2 8121.306} C_VEL
LIN {X 0,Y 258.357,Z 1116.937,A -85,B 0,C 180,E1 8118.971,E2 8118.971} C_VEL
LIN {X 0,Y 242.518,Z 1123.699,A -85,B 0,C 180,E1 8116.282,E2 8116.282} C_VEL
LIN {X 0,Y 226.246,Z 1130.01,A -85,B 0,C 180,E1 8112.507,E2 8112.507} C_VEL
LIN {X 0,Y 212.763,Z 1135.014,A -85,B 0,C 180,E1 8108.105,E2 8108.105} C_VEL
LIN {X 0,Y 201.179,Z 1139.251,A -85,B 0,C 180,E1 8102.505,E2 8102.505} C_VEL
LIN {X 0,Y 192.038,Z 1142.987,A -85,B 0,C 180,E1 8094.922,E2 8094.922} C_VEL
LIN {X 0,Y 187.842,Z 1146.158,A -85,B 0,C 180,E1 8085.512,E2 8085.512} C_VEL
LIN {X 0,Y 190.633,Z 1148.835,A -85,B 0,C 180,E1 8075.156,E2 8075.156} C_VEL
LIN {X 0,Y 200.456,Z 1150.729,A -85,B 0,C 180,E1 8065.691,E2 8065.691} C_VEL
LIN {X 0,Y 212.715,Z 1151.566,A -85,B 0,C 180,E1 8059.187,E2 8059.187} C_VEL
LIN {X 0,Y 201.356,Z 1160.422,A -85,B 0,C 180,E1 8053.261,E2 8053.261} C_VEL
LIN {X 0,Y 191.006,Z 1168.648,A -85,B 0,C 180,E1 8045.899,E2 8045.899} C_VEL
LIN {X 0,Y 184.44,Z 1174.209,A -85,B 0,C 180,E1 8039.207,E2 8039.207} C_VEL
LIN {X 0,Y 179.323,Z 1179.174,A -85,B 0,C 180,E1 8030.911,E2 8030.911} C_VEL
LIN {X 0,Y 177.091,Z 1181.896,A -85,B 0,C 180,E1 8024.055,E2 8024.055} C_VEL
LIN {X 0,Y 176.264,Z 1183.446,A -85,B 0,C 180,E1 8017.829,E2 8017.829} C_VEL
LIN {X 0,Y 176.059,Z 1184.108,A -85,B 0,C 180,E1 8011.957,E2 8011.957} C_VEL
LIN {X 0,Y 176.079,Z 1184.012,A -85,B 0,C 180,E1 8006.423,E2 8006.423} C_VEL
LIN {X 0,Y 176.435,Z 1183.099,A -85,B 0,C 180,E1 8000.215,E2 8000.215} C_VEL
LIN {X 0,Y 178.042,Z 1180.69,A -85,B 0,C 180,E1 7992.351,E2 7992.351} C_VEL
LIN {X 0,Y 181.282,Z 1177.159,A -85,B 0,C 180,E1 7985.221,E2 7985.221} C_VEL
LIN {X 0,Y 186.821,Z 1172.237,A -85,B 0,C 180,E1 7978.009,E2 7978.009} C_VEL
LIN {X 0,Y 195.744,Z 1164.92,A -85,B 0,C 180,E1 7970.324,E2 7970.324} C_VEL
LIN {X 0,Y 206.927,Z 1156.237,A -85,B 0,C 180,E1 7963.553,E2 7963.553} C_VEL
LIN {X 0,Y 220.423,Z 1145.589,A -85,B 0,C 180,E1 7957.46,E2 7957.46} C_VEL
LIN {X 0,Y 236.282,Z 1132.746,A -85,B 0,C 180,E1 7951.936,E2 7951.936} C_VEL
LIN {X 0,Y 252.419,Z 1119.048,A -85,B 0,C 180,E1 7947.47,E2 7947.47} C_VEL
LIN {X 0,Y 267.933,Z 1104.784,A -85,B 0,C 180,E1 7943.901,E2 7943.901} C_VEL
LIN {X 0,Y 283.536,Z 1089.619,A -85,B 0,C 180,E1 7940.858,E2 7940.858} C_VEL
LIN {X 0,Y 298.983,Z 1073.198,A -85,B 0,C 180,E1 7938.245,E2 7938.245} C_VEL
LIN {X 0,Y 315.288,Z 1054.285,A -85,B 0,C 180,E1 7935.827,E2 7935.827} C_VEL
LIN {X 0,Y 328.279,Z 1037.753,A -85,B 0,C 180,E1 7934.103,E2 7934.103} C_VEL
LIN {X 0,Y 342.425,Z 1017.94,A -85,B 0,C 180,E1 7932.393,E2 7932.393} C_VEL
LIN {X 0,Y 354.52,Z 999.225,A -85,B 0,C 180,E1 7931.053,E2 7931.053} C_VEL
LIN {X 0,Y 366.321,Z 978.576,A -85,B 0,C 180,E1 7929.831,E2 7929.831} C_VEL
LIN {X 0,Y 376.095,Z 959.554,A -85,B 0,C 180,E1 7928.87,E2 7928.87} C_VEL
LIN {X 0,Y 386.127,Z 937.015,A -85,B 0,C 180,E1 7927.924,E2 7927.924} C_VEL
LIN {X 0,Y 394.985,Z 913.959,A -85,B 0,C 180,E1 7927.121,E2 7927.121} C_VEL
LIN {X 0,Y 405.584,Z 880.158,A -85,B 0,C 180,E1 7926.191,E2 7926.191} C_VEL
LIN {X 0,Y 417.821,Z 837.614,A -85,B 0,C 180,E1 7925.309,E2 7925.309} C_VEL
LIN {X 0,Y 430.758,Z 788.266,A -85,B 0,C 180,E1 7924.495,E2 7924.495} C_VEL
LIN {X 0,Y 436.685,Z 763.616,A -85,B 0,C 180,E1 7924.099,E2 7924.099} C_VEL
LIN {X 0,Y 429.521,Z 791.933,A -85,B 0,C 180,E1 7921.701,E2 7921.701} C_VEL
LIN {X 0,Y 423.084,Z 818.472,A -85,B 0,C 180,E1 7919.114,E2 7919.114} C_VEL
LIN {X 0,Y 421.513,Z 825.009,A -85,B 0,C 180,E1 7918.583,E2 7918.583} C_VEL
LIN {X 0,Y 416.852,Z 843.111,A -85,B 0,C 180,E1 7917.571,E2 7917.571} C_VEL
LIN {X 0,Y 415.345,Z 849.423,A -85,B 0,C 180,E1 7916.993,E2 7916.993} C_VEL
LIN {X 0,Y 413.492,Z 858.122,A -85,B 0,C 180,E1 7915.905,E2 7915.905} C_VEL
LIN {X 0,Y 400.889,Z 898.411,A -85,B 0,C 180,E1 7915.124,E2 7915.124} C_VEL
LIN {X 0,Y 389.461,Z 931.856,A -85,B 0,C 180,E1 7914.253,E2 7914.253} C_VEL
LIN {X 0,Y 380.386,Z 954.776,A -85,B 0,C 180,E1 7913.499,E2 7913.499} C_VEL
LIN {X 0,Y 369.549,Z 977.907,A -85,B 0,C 180,E1 7912.564,E2 7912.564} C_VEL
LIN {X 0,Y 356.965,Z 1001.263,A -85,B 0,C 180,E1 7911.391,E2 7911.391} C_VEL
LIN {X 0,Y 344.986,Z 1020.998,A -85,B 0,C 180,E1 7910.193,E2 7910.193} C_VEL
LIN {X 0,Y 331.185,Z 1041.183,A -85,B 0,C 180,E1 7908.683,E2 7908.683} C_VEL
LIN {X 0,Y 319.761,Z 1056.449,A -85,B 0,C 180,E1 7907.309,E2 7907.309} C_VEL
LIN {X 0,Y 305.284,Z 1074.294,A -85,B 0,C 180,E1 7905.392,E2 7905.392} C_VEL
LIN {X 0,Y 290.379,Z 1090.811,A -85,B 0,C 180,E1 7903.177,E2 7903.177} C_VEL
LIN {X 0,Y 273.886,Z 1107.684,A -85,B 0,C 180,E1 7900.362,E2 7900.362} C_VEL
LIN {X 0,Y 257.93,Z 1122.57,A -85,B 0,C 180,E1 7897.191,E2 7897.191} C_VEL
LIN {X 0,Y 241.631,Z 1136.578,A -85,B 0,C 180,E1 7893.35,E2 7893.35} C_VEL
LIN {X 0,Y 226.324,Z 1148.946,A -85,B 0,C 180,E1 7888.983,E2 7888.983} C_VEL
LIN {X 0,Y 211.157,Z 1160.321,A -85,B 0,C 180,E1 7883.603,E2 7883.603} C_VEL
LIN {X 0,Y 197.42,Z 1170.288,A -85,B 0,C 180,E1 7877.25,E2 7877.25} C_VEL
LIN {X 0,Y 186.11,Z 1178.477,A -85,B 0,C 180,E1 7870.138,E2 7870.138} C_VEL
LIN {X 0,Y 177.504,Z 1184.922,A -85,B 0,C 180,E1 7862.332,E2 7862.332} C_VEL
LIN {X 0,Y 171.747,Z 1189.812,A -85,B 0,C 180,E1 7853.93,E2 7853.93} C_VEL
LIN {X 0,Y 168.838,Z 1193.163,A -85,B 0,C 180,E1 7845.451,E2 7845.451} C_VEL
LIN {X 0,Y 168.079,Z 1194.799,A -85,B 0,C 180,E1 7838.204,E2 7838.204} C_VEL
LIN {X 0,Y 168.045,Z 1195.414,A -85,B 0,C 180,E1 7832.383,E2 7832.383} C_VEL
LIN {X 0,Y 168.038,Z 1195.376,A -85,B 0,C 180,E1 7826.926,E2 7826.926} C_VEL
LIN {X 0,Y 168.115,Z 1194.632,A -85,B 0,C 180,E1 7820.755,E2 7820.755} C_VEL
LIN {X 0,Y 169.243,Z 1192.56,A -85,B 0,C 180,E1 7812.814,E2 7812.814} C_VEL
LIN {X 0,Y 172.531,Z 1189.096,A -85,B 0,C 180,E1 7804.601,E2 7804.601} C_VEL
LIN {X 0,Y 179.021,Z 1183.709,A -85,B 0,C 180,E1 7796.041,E2 7796.041} C_VEL
LIN {X 0,Y 189.036,Z 1176.275,A -85,B 0,C 180,E1 7787.776,E2 7787.776} C_VEL
LIN {X 0,Y 201.05,Z 1167.675,A -85,B 0,C 180,E1 7780.888,E2 7780.888} C_VEL
LIN {X 0,Y 215.415,Z 1157.122,A -85,B 0,C 180,E1 7774.753,E2 7774.753} C_VEL
LIN {X 0,Y 231.059,Z 1145.057,A -85,B 0,C 180,E1 7769.559,E2 7769.559} C_VEL
LIN {X 0,Y 248.236,Z 1130.942,A -85,B 0,C 180,E1 7764.997,E2 7764.997} C_VEL
LIN {X 0,Y 263.966,Z 1116.935,A -85,B 0,C 180,E1 7761.528,E2 7761.528} C_VEL
LIN {X 0,Y 245.978,Z 1124.596,A -85,B 0,C 180,E1 7758.978,E2 7758.978} C_VEL
LIN {X 0,Y 229.045,Z 1131.046,A -85,B 0,C 180,E1 7755.704,E2 7755.704} C_VEL
LIN {X 0,Y 213.045,Z 1136.678,A -85,B 0,C 180,E1 7751.369,E2 7751.369} C_VEL
LIN {X 0,Y 200.174,Z 1141.044,A -85,B 0,C 180,E1 7746.309,E2 7746.309} C_VEL
LIN {X 0,Y 189.989,Z 1144.548,A -85,B 0,C 180,E1 7740.138,E2 7740.138} C_VEL
LIN {X 0,Y 182.83,Z 1147.663,A -85,B 0,C 180,E1 7732.142,E2 7732.142} C_VEL
LIN {X 0,Y 180.563,Z 1150.391,A -85,B 0,C 180,E1 7722.6,E2 7722.6} C_VEL
LIN {X 0,Y 187.117,Z 1153.056,A -85,B 0,C 180,E1 7710.201,E2 7710.201} C_VEL
LIN {X 0,Y 199.332,Z 1154.296,A -85,B 0,C 180,E1 7701.537,E2 7701.537} C_VEL
LIN {X 0,Y 203.796,Z 1154.589,A -85,B 0,C 180,E1 7699.295,E2 7699.295} C_VEL
LIN {X 0,Y 190.817,Z 1164.143,A -85,B 0,C 180,E1 7692.127,E2 7692.127} C_VEL
LIN {X 0,Y 181.872,Z 1170.879,A -85,B 0,C 180,E1 7685.262,E2 7685.262} C_VEL
LIN {X 0,Y 174.555,Z 1176.795,A -85,B 0,C 180,E1 7676.91,E2 7676.91} C_VEL
LIN {X 0,Y 170.815,Z 1180.321,A -85,B 0,C 180,E1 7669.851,E2 7669.851} C_VEL
LIN {X 0,Y 168.72,Z 1182.992,A -85,B 0,C 180,E1 7661.975,E2 7661.975} C_VEL
LIN {X 0,Y 168.114,Z 1184.21,A -85,B 0,C 180,E1 7654.781,E2 7654.781} C_VEL
LIN {X 0,Y 168.061,Z 1184.421,A -85,B 0,C 180,E1 7648.641,E2 7648.641} C_VEL
LIN {X 0,Y 168.24,Z 1183.859,A -85,B 0,C 180,E1 7642.491,E2 7642.491} C_VEL
LIN {X 0,Y 169.072,Z 1182.398,A -85,B 0,C 180,E1 7635.907,E2 7635.907} C_VEL
LIN {X 0,Y 171.199,Z 1179.955,A -85,B 0,C 180,E1 7629.133,E2 7629.133} C_VEL
LIN {X 0,Y 176.172,Z 1175.534,A -85,B 0,C 180,E1 7620.789,E2 7620.789} C_VEL
LIN {X 0,Y 183.533,Z 1169.652,A -85,B 0,C 180,E1 7613.187,E2 7613.187} C_VEL
LIN {X 0,Y 194.119,Z 1161.819,A -85,B 0,C 180,E1 7605.724,E2 7605.724} C_VEL
LIN {X 0,Y 206.682,Z 1152.526,A -85,B 0,C 180,E1 7599.288,E2 7599.288} C_VEL
LIN {X 0,Y 222.345,Z 1140.7,A -85,B 0,C 180,E1 7593.24,E2 7593.24} C_VEL
LIN {X 0,Y 237.858,Z 1128.498,A -85,B 0,C 180,E1 7588.536,E2 7588.536} C_VEL
LIN {X 0,Y 253.916,Z 1114.859,A -85,B 0,C 180,E1 7584.552,E2 7584.552} C_VEL
LIN {X 0,Y 270.208,Z 1100.201,A -85,B 0,C 180,E1 7581.18,E2 7581.18} C_VEL
LIN {X 0,Y 285.622,Z 1085.087,A -85,B 0,C 180,E1 7578.442,E2 7578.442} C_VEL
LIN {X 0,Y 302.88,Z 1066.68,A -85,B 0,C 180,E1 7575.79,E2 7575.79} C_VEL
LIN {X 0,Y 318.501,Z 1048.457,A -85,B 0,C 180,E1 7573.693,E2 7573.693} C_VEL
LIN {X 0,Y 332.235,Z 1030.468,A -85,B 0,C 180,E1 7572.023,E2 7572.023} C_VEL
LIN {X 0,Y 344.423,Z 1013.261,A -85,B 0,C 180,E1 7570.673,E2 7570.673} C_VEL
LIN {X 0,Y 357.219,Z 992.871,A -85,B 0,C 180,E1 7569.343,E2 7569.343} C_VEL
LIN {X 0,Y 369.208,Z 971.621,A -85,B 0,C 180,E1 7568.191,E2 7568.191} C_VEL
LIN {X 0,Y 379.938,Z 949.482,A -85,B 0,C 180,E1 7567.203,E2 7567.203} C_VEL
LIN {X 0,Y 390.03,Z 925.278,A -85,B 0,C 180,E1 7566.31,E2 7566.31} C_VEL
LIN {X 0,Y 398.289,Z 901.807,A -85,B 0,C 180,E1 7565.6,E2 7565.6} C_VEL
LIN {X 0,Y 410.933,Z 860.146,A -85,B 0,C 180,E1 7564.618,E2 7564.618} C_VEL
LIN {X 0,Y 424.001,Z 813.56,A -85,B 0,C 180,E1 7563.819,E2 7563.819} C_VEL
LIN {X 0,Y 430.813,Z 787.165,A -85,B 0,C 180,E1 7563.402,E2 7563.402} C_VEL
LIN {X 0,Y 423.902,Z 813.641,A -85,B 0,C 180,E1 7560.929,E2 7560.929} C_VEL
LIN {X 0,Y 418.546,Z 835.306,A -85,B 0,C 180,E1 7558.631,E2 7558.631} C_VEL
LIN {X 0,Y 415.345,Z 849.423,A -85,B 0,C 180,E1 7556.993,E2 7556.993} C_VEL
LIN {X 0,Y 414.5,Z 853.045,A -85,B 0,C 180,E1 7556.679,E2 7556.679} C_VEL
LIN {X 0,Y 412.719,Z 859.248,A -85,B 0,C 180,E1 7556.465,E2 7556.465} C_VEL
LIN {X 0,Y 409.99,Z 867.954,A -85,B 0,C 180,E1 7556.481,E2 7556.481} C_VEL
LIN {X 0,Y 405.875,Z 880.33,A -85,B 0,C 180,E1 7556.609,E2 7556.609} C_VEL
LIN {X 0,Y 404.829,Z 883.706,A -85,B 0,C 180,E1 7556.572,E2 7556.572} C_VEL
LIN {X 0,Y 392.043,Z 922.239,A -85,B 0,C 180,E1 7555.698,E2 7555.698} C_VEL
LIN {X 0,Y 383.374,Z 944.762,A -85,B 0,C 180,E1 7555.042,E2 7555.042} C_VEL
LIN {X 0,Y 373.808,Z 966.639,A -85,B 0,C 180,E1 7554.271,E2 7554.271} C_VEL
LIN {X 0,Y 362.412,Z 988.842,A -85,B 0,C 180,E1 7553.307,E2 7553.307} C_VEL
LIN {X 0,Y 349.259,Z 1011.499,A -85,B 0,C 180,E1 7552.1,E2 7552.1} C_VEL
LIN {X 0,Y 336.57,Z 1030.816,A -85,B 0,C 180,E1 7550.842,E2 7550.842} C_VEL
LIN {X 0,Y 321.63,Z 1051.167,A -85,B 0,C 180,E1 7549.214,E2 7549.214} C_VEL
LIN {X 0,Y 309.051,Z 1066.747,A -85,B 0,C 180,E1 7547.694,E2 7547.694} C_VEL
LIN {X 0,Y 293.63,Z 1084.339,A -85,B 0,C 180,E1 7545.606,E2 7545.606} C_VEL
LIN {X 0,Y 278.684,Z 1099.705,A -85,B 0,C 180,E1 7543.318,E2 7543.318} C_VEL
LIN {X 0,Y 262.953,Z 1114.77,A -85,B 0,C 180,E1 7540.556,E2 7540.556} C_VEL
LIN {X 0,Y 246.303,Z 1129.23,A -85,B 0,C 180,E1 7537.141,E2 7537.141} C_VEL
LIN {X 0,Y 229.126,Z 1143.012,A -85,B 0,C 180,E1 7532.895,E2 7532.895} C_VEL
LIN {X 0,Y 213.136,Z 1155.054,A -85,B 0,C 180,E1 7527.986,E2 7527.986} C_VEL
LIN {X 0,Y 197.88,Z 1165.74,A -85,B 0,C 180,E1 7522.017,E2 7522.017} C_VEL
LIN {X 0,Y 184.743,Z 1174.692,A -85,B 0,C 180,E1 7515.149,E2 7515.149} C_VEL
LIN {X 0,Y 174.24,Z 1181.971,A -85,B 0,C 180,E1 7507.46,E2 7507.46} C_VEL
LIN {X 0,Y 166.431,Z 1187.713,A -85,B 0,C 180,E1 7498.721,E2 7498.721} C_VEL
LIN {X 0,Y 161.982,Z 1191.661,A -85,B 0,C 180,E1 7489.842,E2 7489.842} C_VEL
LIN {X 0,Y 160.277,Z 1194.021,A -85,B 0,C 180,E1 7481.636,E2 7481.636} C_VEL
LIN {X 0,Y 160.033,Z 1195.038,A -85,B 0,C 180,E1 7474.654,E2 7474.654} C_VEL
LIN {X 0,Y 160.059,Z 1195.219,A -85,B 0,C 180,E1 7468.922,E2 7468.922} C_VEL
LIN {X 0,Y 160.067,Z 1194.687,A -85,B 0,C 180,E1 7462.458,E2 7462.458} C_VEL
LIN {X 0,Y 160.695,Z 1193.235,A -85,B 0,C 180,E1 7455.215,E2 7455.215} C_VEL
LIN {X 0,Y 163.576,Z 1190.094,A -85,B 0,C 180,E1 7446.202,E2 7446.202} C_VEL
LIN {X 0,Y 169.335,Z 1185.477,A -85,B 0,C 180,E1 7437.493,E2 7437.493} C_VEL
LIN {X 0,Y 178.519,Z 1178.919,A -85,B 0,C 180,E1 7429.052,E2 7429.052} C_VEL
LIN {X 0,Y 191.164,Z 1170.297,A -85,B 0,C 180,E1 7421.227,E2 7421.227} C_VEL
LIN {X 0,Y 205.96,Z 1160.039,A -85,B 0,C 180,E1 7414.612,E2 7414.612} C_VEL
LIN {X 0,Y 222.085,Z 1148.365,A -85,B 0,C 180,E1 7409.134,E2 7409.134} C_VEL
LIN {X 0,Y 238.704,Z 1135.376,A -85,B 0,C 180,E1 7404.631,E2 7404.631} C_VEL
LIN {X 0,Y 251.33,Z 1124.821,A -85,B 0,C 180,E1 7401.715,E2 7401.715} C_VEL
LIN {X 0,Y 233.862,Z 1131.507,A -85,B 0,C 180,E1 7398.962,E2 7398.962} C_VEL
LIN {X 0,Y 216.552,Z 1137.461,A -85,B 0,C 180,E1 7395.19,E2 7395.19} C_VEL
LIN {X 0,Y 201.626,Z 1142.272,A -85,B 0,C 180,E1 7390.573,E2 7390.573} C_VEL
LIN {X 0,Y 188.577,Z 1146.331,A -85,B 0,C 180,E1 7384.529,E2 7384.529} C_VEL
LIN {X 0,Y 178.138,Z 1149.889,A -85,B 0,C 180,E1 7376.138,E2 7376.138} C_VEL
LIN {X 0,Y 173.32,Z 1152.86,A -85,B 0,C 180,E1 7365.637,E2 7365.637} C_VEL
LIN {X 0,Y 176.378,Z 1155.309,A -85,B 0,C 180,E1 7354.118,E2 7354.118} C_VEL
LIN {X 0,Y 186.507,Z 1156.908,A -85,B 0,C 180,E1 7344.242,E2 7344.242} C_VEL
LIN {X 0,Y 194.842,Z 1157.525,A -85,B 0,C 180,E1 7339.425,E2 7339.425} C_VEL
LIN {X 0,Y 182.462,Z 1166.063,A -85,B 0,C 180,E1 7332.384,E2 7332.384} C_VEL
LIN {X 0,Y 171.903,Z 1173.567,A -85,B 0,C 180,E1 7323.718,E2 7323.718} C_VEL
LIN {X 0,Y 165.84,Z 1178.237,A -85,B 0,C 180,E1 7316.056,E2 7316.056} C_VEL
LIN {X 0,Y 161.877,Z 1181.928,A -85,B 0,C 180,E1 7307.251,E2 7307.251} C_VEL
LIN {X 0,Y 160.438,Z 1183.791,A -85,B 0,C 180,E1 7299.692,E2 7299.692} C_VEL
LIN {X 0,Y 160.088,Z 1184.552,A -85,B 0,C 180,E1 7293.585,E2 7293.585} C_VEL
LIN {X 0,Y 160.069,Z 1184.643,A -85,B 0,C 180,E1 7287.856,E2 7287.856} C_VEL
LIN {X 0,Y 160.295,Z 1184.067,A -85,B 0,C 180,E1 7281.756,E2 7281.756} C_VEL
LIN {X 0,Y 161.28,Z 1182.592,A -85,B 0,C 180,E1 7274.912,E2 7274.912} C_VEL
LIN {X 0,Y 163.905,Z 1179.953,A -85,B 0,C 180,E1 7267.403,E2 7267.403} C_VEL
LIN {X 0,Y 169.857,Z 1175.14,A -85,B 0,C 180,E1 7258.41,E2 7258.41} C_VEL
LIN {X 0,Y 177.806,Z 1169.373,A -85,B 0,C 180,E1 7250.9,E2 7250.9} C_VEL
LIN {X 0,Y 189.992,Z 1160.916,A -85,B 0,C 180,E1 7242.992,E2 7242.992} C_VEL
LIN {X 0,Y 203.893,Z 1151.267,A -85,B 0,C 180,E1 7236.469,E2 7236.469} C_VEL
LIN {X 0,Y 219.225,Z 1140.072,A -85,B 0,C 180,E1 7230.974,E2 7230.974} C_VEL
LIN {X 0,Y 235.457,Z 1127.71,A -85,B 0,C 180,E1 7226.367,E2 7226.367} C_VEL
LIN {X 0,Y 252.148,Z 1114.031,A -85,B 0,C 180,E1 7222.498,E2 7222.498} C_VEL
LIN {X 0,Y 269.788,Z 1098.361,A -85,B 0,C 180,E1 7219.087,E2 7219.087} C_VEL
LIN {X 0,Y 286.532,Z 1082.31,A -85,B 0,C 180,E1 7216.344,E2 7216.344} C_VEL
LIN {X 0,Y 301.26,Z 1066.606,A -85,B 0,C 180,E1 7214.218,E2 7214.218} C_VEL
LIN {X 0,Y 316.668,Z 1049.025,A -85,B 0,C 180,E1 7212.258,E2 7212.258} C_VEL
LIN {X 0,Y 332.003,Z 1029.298,A -85,B 0,C 180,E1 7210.497,E2 7210.497} C_VEL
LIN {X 0,Y 346.811,Z 1008.088,A -85,B 0,C 180,E1 7208.957,E2 7208.957} C_VEL
LIN {X 0,Y 359.238,Z 988.19,A -85,B 0,C 180,E1 7207.766,E2 7207.766} C_VEL
LIN {X 0,Y 370.969,Z 966.616,A -85,B 0,C 180,E1 7206.693,E2 7206.693} C_VEL
LIN {X 0,Y 381.39,Z 944.895,A -85,B 0,C 180,E1 7205.797,E2 7205.797} C_VEL
LIN {X 0,Y 389.965,Z 923.784,A -85,B 0,C 180,E1 7205.071,E2 7205.071} C_VEL
LIN {X 0,Y 398.114,Z 900.522,A -85,B 0,C 180,E1 7204.406,E2 7204.406} C_VEL
LIN {X 0,Y 410.422,Z 860.631,A -85,B 0,C 180,E1 7203.504,E2 7203.504} C_VEL
LIN {X 0,Y 422.872,Z 817.117,A -85,B 0,C 180,E1 7202.787,E2 7202.787} C_VEL
LIN {X 0,Y 424.89,Z 809.584,A -85,B 0,C 180,E1 7202.652,E2 7202.652} C_VEL
LIN {X 0,Y 417.777,Z 836.426,A -85,B 0,C 180,E1 7199.897,E2 7199.897} C_VEL
LIN {X 0,Y 411.868,Z 860.519,A -85,B 0,C 180,E1 7197.043,E2 7197.043} C_VEL
LIN {X 0,Y 411.517,Z 861.865,A -85,B 0,C 180,E1 7196.954,E2 7196.954} C_VEL
LIN {X 0,Y 404.829,Z 883.706,A -85,B 0,C 180,E1 7196.572,E2 7196.572} C_VEL
LIN {X 0,Y 402.421,Z 891.093,A -85,B 0,C 180,E1 7196.567,E2 7196.567} C_VEL
LIN {X 0,Y 395.232,Z 910.797,A -85,B 0,C 180,E1 7197.038,E2 7197.038} C_VEL
LIN {X 0,Y 393.068,Z 917.075,A -85,B 0,C 180,E1 7197.001,E2 7197.001} C_VEL
LIN {X 0,Y 384.695,Z 939.343,A -85,B 0,C 180,E1 7196.407,E2 7196.407} C_VEL
LIN {X 0,Y 376.937,Z 957.356,A -85,B 0,C 180,E1 7195.832,E2 7195.832} C_VEL
LIN {X 0,Y 366.938,Z 978.199,A -85,B 0,C 180,E1 7195.048,E2 7195.048} C_VEL
LIN {X 0,Y 354.856,Z 999.784,A -85,B 0,C 180,E1 7194.048,E2 7194.048} C_VEL
LIN {X 0,Y 341.598,Z 1021.051,A -85,B 0,C 180,E1 7192.854,E2 7192.854} C_VEL
LIN {X 0,Y 327.105,Z 1041.496,A -85,B 0,C 180,E1 7191.423,E2 7191.423} C_VEL
LIN {X 0,Y 310.719,Z 1062.156,A -85,B 0,C 180,E1 7189.618,E2 7189.618} C_VEL
LIN {X 0,Y 297.276,Z 1077.545,A -85,B 0,C 180,E1 7187.963,E2 7187.963} C_VEL
LIN {X 0,Y 280.703,Z 1094.898,A -85,B 0,C 180,E1 7185.657,E2 7185.657} C_VEL
LIN {X 0,Y 266.116,Z 1108.758,A -85,B 0,C 180,E1 7183.348,E2 7183.348} C_VEL
LIN {X 0,Y 249.556,Z 1123.429,A -85,B 0,C 180,E1 7180.306,E2 7180.306} C_VEL
LIN {X 0,Y 232.201,Z 1137.389,A -85,B 0,C 180,E1 7176.511,E2 7176.511} C_VEL
LIN {X 0,Y 215.208,Z 1149.97,A -85,B 0,C 180,E1 7171.97,E2 7171.97} C_VEL
LIN {X 0,Y 199.641,Z 1160.843,A -85,B 0,C 180,E1 7166.755,E2 7166.755} C_VEL
LIN {X 0,Y 184.716,Z 1170.603,A -85,B 0,C 180,E1 7160.227,E2 7160.227} C_VEL
LIN {X 0,Y 171.818,Z 1178.868,A -85,B 0,C 180,E1 7152.452,E2 7152.452} C_VEL
LIN {X 0,Y 162.358,Z 1185.186,A -85,B 0,C 180,E1 7144.08,E2 7144.08} C_VEL
LIN {X 0,Y 156.237,Z 1189.655,A -85,B 0,C 180,E1 7135.385,E2 7135.385} C_VEL
LIN {X 0,Y 152.898,Z 1192.87,A -85,B 0,C 180,E1 7125.937,E2 7125.937} C_VEL
LIN {X 0,Y 152.087,Z 1194.37,A -85,B 0,C 180,E1 7118.312,E2 7118.312} C_VEL
LIN {X 0,Y 152.058,Z 1194.927,A -85,B 0,C 180,E1 7111.789,E2 7111.789} C_VEL
LIN {X 0,Y 152.038,Z 1194.81,A -85,B 0,C 180,E1 7105.847,E2 7105.847} C_VEL
LIN {X 0,Y 152.251,Z 1193.921,A -85,B 0,C 180,E1 7098.633,E2 7098.633} C_VEL
LIN {X 0,Y 154.019,Z 1191.616,A -85,B 0,C 180,E1 7089.87,E2 7089.87} C_VEL
LIN {X 0,Y 158.886,Z 1187.62,A -85,B 0,C 180,E1 7080.28,E2 7080.28} C_VEL
LIN {X 0,Y 166.907,Z 1182.076,A -85,B 0,C 180,E1 7071.457,E2 7071.457} C_VEL
LIN {X 0,Y 178.413,Z 1174.605,A -85,B 0,C 180,E1 7063.229,E2 7063.229} C_VEL
LIN {X 0,Y 192.811,Z 1165.264,A -85,B 0,C 180,E1 7055.997,E2 7055.997} C_VEL
LIN {X 0,Y 208.94,Z 1154.392,A -85,B 0,C 180,E1 7049.977,E2 7049.977} C_VEL
LIN {X 0,Y 226.152,Z 1141.881,A -85,B 0,C 180,E1 7044.986,E2 7044.986} C_VEL
LIN {X 0,Y 238.822,Z 1132.041,A -85,B 0,C 180,E1 7041.878,E2 7041.878} C_VEL
LIN {X 0,Y 220.545,Z 1138.271,A -85,B 0,C 180,E1 7038.632,E2 7038.632} C_VEL
LIN {X 0,Y 203.14,Z 1143.653,A -85,B 0,C 180,E1 7034.247,E2 7034.247} C_VEL
LIN {X 0,Y 188.556,Z 1147.896,A -85,B 0,C 180,E1 7028.846,E2 7028.846} C_VEL
LIN {X 0,Y 177.107,Z 1151.199,A -85,B 0,C 180,E1 7022.265,E2 7022.265} C_VEL
LIN {X 0,Y 168.785,Z 1154.121,A -85,B 0,C 180,E1 7013.537,E2 7013.537} C_VEL
LIN {X 0,Y 165.855,Z 1156.675,A -85,B 0,C 180,E1 7002.818,E2 7002.818} C_VEL
LIN {X 0,Y 172.476,Z 1159.036,A -85,B 0,C 180,E1 6989.325,E2 6989.325} C_VEL
LIN {X 0,Y 185.656,Z 1160.159,A -85,B 0,C 180,E1 6979.738,E2 6979.738} C_VEL
LIN {X 0,Y 185.767,Z 1160.271,A -85,B 0,C 180,E1 6979.521,E2 6979.521} C_VEL
LIN {X 0,Y 173.208,Z 1168.545,A -85,B 0,C 180,E1 6972.044,E2 6972.044} C_VEL
LIN {X 0,Y 163.562,Z 1174.913,A -85,B 0,C 180,E1 6963.757,E2 6963.757} C_VEL
LIN {X 0,Y 156.801,Z 1179.885,A -85,B 0,C 180,E1 6954.492,E2 6954.492} C_VEL
LIN {X 0,Y 153.567,Z 1182.711,A -85,B 0,C 180,E1 6946.263,E2 6946.263} C_VEL
LIN {X 0,Y 152.375,Z 1184.24,A -85,B 0,C 180,E1 6939.066,E2 6939.066} C_VEL
LIN {X 0,Y 152.077,Z 1184.875,A -85,B 0,C 180,E1 6932.643,E2 6932.643} C_VEL
LIN {X 0,Y 152.081,Z 1184.866,A -85,B 0,C 180,E1 6926.99,E2 6926.99} C_VEL
LIN {X 0,Y 152.403,Z 1184.213,A -85,B 0,C 180,E1 6920.564,E2 6920.564} C_VEL
LIN {X 0,Y 153.647,Z 1182.662,A -85,B 0,C 180,E1 6913.366,E2 6913.366} C_VEL
LIN {X 0,Y 157.369,Z 1179.511,A -85,B 0,C 180,E1 6904.407,E2 6904.407} C_VEL
LIN {X 0,Y 164.187,Z 1174.53,A -85,B 0,C 180,E1 6895.509,E2 6895.509} C_VEL
LIN {X 0,Y 174.003,Z 1168.078,A -85,B 0,C 180,E1 6887.313,E2 6887.313} C_VEL
LIN {X 0,Y 186.584,Z 1159.818,A -85,B 0,C 180,E1 6879.982,E2 6879.982} C_VEL
LIN {X 0,Y 202.513,Z 1149.202,A -85,B 0,C 180,E1 6873.234,E2 6873.234} C_VEL
LIN {X 0,Y 218.604,Z 1138.013,A -85,B 0,C 180,E1 6868.029,E2 6868.029} C_VEL
LIN {X 0,Y 235.71,Z 1125.156,A -85,B 0,C 180,E1 6863.621,E2 6863.621} C_VEL
LIN {X 0,Y 253.943,Z 1110.442,A -85,B 0,C 180,E1 6859.793,E2 6859.793} C_VEL
LIN {X 0,Y 268.89,Z 1097.277,A -85,B 0,C 180,E1 6857.135,E2 6857.135} C_VEL
LIN {X 0,Y 285.295,Z 1081.796,A -85,B 0,C 180,E1 6854.616,E2 6854.616} C_VEL
LIN {X 0,Y 300.176,Z 1066.285,A -85,B 0,C 180,E1 6852.597,E2 6852.597} C_VEL
LIN {X 0,Y 315.818,Z 1048.552,A -85,B 0,C 180,E1 6850.715,E2 6850.715} C_VEL
LIN {X 0,Y 330.62,Z 1029.924,A -85,B 0,C 180,E1 6849.113,E2 6849.113} C_VEL
LIN {X 0,Y 345.422,Z 1009.043,A -85,B 0,C 180,E1 6847.652,E2 6847.652} C_VEL
LIN {X 0,Y 358.711,Z 988.009,A -85,B 0,C 180,E1 6846.447,E2 6846.447} C_VEL
LIN {X 0,Y 369.639,Z 968.091,A -85,B 0,C 180,E1 6845.494,E2 6845.494} C_VEL
LIN {X 0,Y 380.182,Z 946.531,A -85,B 0,C 180,E1 6844.632,E2 6844.632} C_VEL
LIN {X 0,Y 388.504,Z 926.442,A -85,B 0,C 180,E1 6843.96,E2 6843.96} C_VEL
LIN {X 0,Y 396.122,Z 905.609,A -85,B 0,C 180,E1 6843.368,E2 6843.368} C_VEL
LIN {X 0,Y 409,Z 864.818,A -85,B 0,C 180,E1 6842.458,E2 6842.458} C_VEL
LIN {X 0,Y 419.066,Z 830.712,A -85,B 0,C 180,E1 6841.88,E2 6841.88} C_VEL
LIN {X 0,Y 411.472,Z 859.08,A -85,B 0,C 180,E1 6838.677,E2 6838.677} C_VEL
LIN {X 0,Y 410.085,Z 864.652,A -85,B 0,C 180,E1 6838.027,E2 6838.027} C_VEL
LIN {X 0,Y 397.626,Z 903.577,A -85,B 0,C 180,E1 6837.309,E2 6837.309} C_VEL
LIN {X 0,Y 393.068,Z 917.075,A -85,B 0,C 180,E1 6837.001,E2 6837.001} C_VEL
LIN {X 0,Y 390.483,Z 924.402,A -85,B 0,C 180,E1 6836.968,E2 6836.968} C_VEL
LIN {X 0,Y 382.806,Z 942.814,A -85,B 0,C 180,E1 6837.363,E2 6837.363} C_VEL
LIN {X 0,Y 379.569,Z 949.843,A -85,B 0,C 180,E1 6837.3,E2 6837.3} C_VEL
LIN {X 0,Y 370.571,Z 968.865,A -85,B 0,C 180,E1 6836.659,E2 6836.659} C_VEL
LIN {X 0,Y 360.856,Z 987.401,A -85,B 0,C 180,E1 6835.922,E2 6835.922} C_VEL
LIN {X 0,Y 347.89,Z 1009.163,A -85,B 0,C 180,E1 6834.866,E2 6834.866} C_VEL
LIN {X 0,Y 335.896,Z 1027.112,A -85,B 0,C 180,E1 6833.823,E2 6833.823} C_VEL
LIN {X 0,Y 319.852,Z 1048.692,A -85,B 0,C 180,E1 6832.273,E2 6832.273} C_VEL
LIN {X 0,Y 303.763,Z 1068.032,A -85,B 0,C 180,E1 6830.527,E2 6830.527} C_VEL
LIN {X 0,Y 287.22,Z 1085.747,A -85,B 0,C 180,E1 6828.498,E2 6828.498} C_VEL
LIN {X 0,Y 270.791,Z 1101.964,A -85,B 0,C 180,E1 6826.182,E2 6826.182} C_VEL
LIN {X 0,Y 254.394,Z 1116.438,A -85,B 0,C 180,E1 6823.531,E2 6823.531} C_VEL
LIN {X 0,Y 237.777,Z 1130.182,A -85,B 0,C 180,E1 6820.371,E2 6820.371} C_VEL
LIN {X 0,Y 220.377,Z 1143.154,A -85,B 0,C 180,E1 6816.411,E2 6816.411} C_VEL
LIN {X 0,Y 202.7,Z 1155.399,A -85,B 0,C 180,E1 6811.399,E2 6811.399} C_VEL
LIN {X 0,Y 187.327,Z 1165.348,A -85,B 0,C 180,E1 6805.818,E2 6805.818} C_VEL
LIN {X 0,Y 172.74,Z 1174.283,A -85,B 0,C 180,E1 6798.8,E2 6798.8} C_VEL
LIN {X 0,Y 160.436,Z 1181.762,A -85,B 0,C 180,E1 6790.397,E2 6790.397} C_VEL
LIN {X 0,Y 151.785,Z 1187.302,A -85,B 0,C 180,E1 6781.354,E2 6781.354} C_VEL
LIN {X 0,Y 146.468,Z 1191.216,A -85,B 0,C 180,E1 6771.626,E2 6771.626} C_VEL
LIN {X 0,Y 144.341,Z 1193.6,A -85,B 0,C 180,E1 6762.379,E2 6762.379} C_VEL
LIN {X 0,Y 144.04,Z 1194.527,A -85,B 0,C 180,E1 6754.773,E2 6754.773} C_VEL
LIN {X 0,Y 144.063,Z 1194.676,A -85,B 0,C 180,E1 6748.404,E2 6748.404} C_VEL
LIN {X 0,Y 144.092,Z 1194.152,A -85,B 0,C 180,E1 6741.616,E2 6741.616} C_VEL
LIN {X 0,Y 145.008,Z 1192.639,A -85,B 0,C 180,E1 6733.43,E2 6733.43} C_VEL
LIN {X 0,Y 148.727,Z 1189.401,A -85,B 0,C 180,E1 6723.401,E2 6723.401} C_VEL
LIN {X 0,Y 155.879,Z 1184.62,A -85,B 0,C 180,E1 6713.829,E2 6713.829} C_VEL
LIN {X 0,Y 166.676,Z 1177.918,A -85,B 0,C 180,E1 6704.932,E2 6704.932} C_VEL
LIN {X 0,Y 180.693,Z 1169.382,A -85,B 0,C 180,E1 6697.097,E2 6697.097} C_VEL
LIN {X 0,Y 197.029,Z 1159.083,A -85,B 0,C 180,E1 6690.497,E2 6690.497} C_VEL
LIN {X 0,Y 214.651,Z 1147.195,A -85,B 0,C 180,E1 6685.081,E2 6685.081} C_VEL
LIN {X 0,Y 226.523,Z 1138.579,A -85,B 0,C 180,E1 6682.037,E2 6682.037} C_VEL
LIN {X 0,Y 207.579,Z 1144.368,A -85,B 0,C 180,E1 6678.246,E2 6678.246} C_VEL
LIN {X 0,Y 191.345,Z 1148.875,A -85,B 0,C 180,E1 6673.589,E2 6673.589} C_VEL
LIN {X 0,Y 177.116,Z 1152.629,A -85,B 0,C 180,E1 6667.461,E2 6667.461} C_VEL
LIN {X 0,Y 165.996,Z 1155.665,A -85,B 0,C 180,E1 6659.562,E2 6659.562} C_VEL
LIN {X 0,Y 158.73,Z 1158.772,A -85,B 0,C 180,E1 6647.263,E2 6647.263} C_VEL
LIN {X 0,Y 161.521,Z 1161.158,A -85,B 0,C 180,E1 6633.531,E2 6633.531} C_VEL
LIN {X 0,Y 172.97,Z 1162.582,A -85,B 0,C 180,E1 6622.211,E2 6622.211} C_VEL
LIN {X 0,Y 176.912,Z 1162.865,A -85,B 0,C 180,E1 6619.735,E2 6619.735} C_VEL
LIN {X 0,Y 163.925,Z 1170.752,A -85,B 0,C 180,E1 6611.677,E2 6611.677} C_VEL
LIN {X 0,Y 154.45,Z 1176.765,A -85,B 0,C 180,E1 6602.948,E2 6602.948} C_VEL
LIN {X 0,Y 148.158,Z 1181.029,A -85,B 0,C 180,E1 6593.469,E2 6593.469} C_VEL
LIN {X 0,Y 145.194,Z 1183.597,A -85,B 0,C 180,E1 6584.767,E2 6584.767} C_VEL
LIN {X 0,Y 144.194,Z 1184.966,A -85,B 0,C 180,E1 6576.375,E2 6576.375} C_VEL
LIN {X 0,Y 144.07,Z 1185.252,A -85,B 0,C 180,E1 6569.21,E2 6569.21} C_VEL
LIN {X 0,Y 144.281,Z 1184.78,A -85,B 0,C 180,E1 6562.038,E2 6562.038} C_VEL
LIN {X 0,Y 145.445,Z 1183.337,A -85,B 0,C 180,E1 6554.044,E2 6554.044} C_VEL
LIN {X 0,Y 148.493,Z 1180.806,A -85,B 0,C 180,E1 6545.754,E2 6545.754} C_VEL
LIN {X 0,Y 155.033,Z 1176.406,A -85,B 0,C 180,E1 6536.304,E2 6536.304} C_VEL
LIN {X 0,Y 164.346,Z 1170.555,A -85,B 0,C 180,E1 6527.924,E2 6527.924} C_VEL
LIN {X 0,Y 177.354,Z 1162.643,A -85,B 0,C 180,E1 6519.945,E2 6519.945} C_VEL
LIN {X 0,Y 191.183,Z 1153.999,A -85,B 0,C 180,E1 6513.747,E2 6513.747} C_VEL
LIN {X 0,Y 208.243,Z 1142.841,A -85,B 0,C 180,E1 6507.943,E2 6507.943} C_VEL
LIN {X 0,Y 226.224,Z 1130.327,A -85,B 0,C 180,E1 6503.18,E2 6503.18} C_VEL
LIN {X 0,Y 242.989,Z 1117.491,A -85,B 0,C 180,E1 6499.566,E2 6499.566} C_VEL
LIN {X 0,Y 260.566,Z 1103.125,A -85,B 0,C 180,E1 6496.406,E2 6496.406} C_VEL
LIN {X 0,Y 277.034,Z 1088.251,A -85,B 0,C 180,E1 6493.872,E2 6493.872} C_VEL
LIN {X 0,Y 294.413,Z 1071.124,A -85,B 0,C 180,E1 6491.559,E2 6491.559} C_VEL
LIN {X 0,Y 309.921,Z 1054.337,A -85,B 0,C 180,E1 6489.745,E2 6489.745} C_VEL
LIN {X 0,Y 326.154,Z 1034.718,A -85,B 0,C 180,E1 6488.041,E2 6488.041} C_VEL
LIN {X 0,Y 340.743,Z 1015.134,A -85,B 0,C 180,E1 6486.658,E2 6486.658} C_VEL
LIN {X 0,Y 353.151,Z 996.195,A -85,B 0,C 180,E1 6485.553,E2 6485.553} C_VEL
LIN {X 0,Y 365.229,Z 975.794,A -85,B 0,C 180,E1 6484.554,E2 6484.554} C_VEL
LIN {X 0,Y 375.246,Z 956.228,A -85,B 0,C 180,E1 6483.755,E2 6483.755} C_VEL
LIN {X 0,Y 384.486,Z 936.107,A -85,B 0,C 180,E1 6483.057,E2 6483.057} C_VEL
LIN {X 0,Y 393.034,Z 913.703,A -85,B 0,C 180,E1 6482.403,E2 6482.403} C_VEL
LIN {X 0,Y 405.582,Z 875.921,A -85,B 0,C 180,E1 6481.539,E2 6481.539} C_VEL
LIN {X 0,Y 413.353,Z 850.643,A -85,B 0,C 180,E1 6481.078,E2 6481.078} C_VEL
LIN {X 0,Y 408.631,Z 867.653,A -85,B 0,C 180,E1 6479.102,E2 6479.102} C_VEL
LIN {X 0,Y 395.597,Z 907.916,A -85,B 0,C 180,E1 6478.375,E2 6478.375} C_VEL
LIN {X 0,Y 386.235,Z 933.926,A -85,B 0,C 180,E1 6477.758,E2 6477.758} C_VEL
LIN {X 0,Y 379.569,Z 949.843,A -85,B 0,C 180,E1 6477.3,E2 6477.3} C_VEL
LIN {X 0,Y 376.193,Z 957.123,A -85,B 0,C 180,E1 6477.226,E2 6477.226} C_VEL
LIN {X 0,Y 366.938,Z 974.933,A -85,B 0,C 180,E1 6477.544,E2 6477.544} C_VEL
LIN {X 0,Y 363.273,Z 981.361,A -85,B 0,C 180,E1 6477.447,E2 6477.447} C_VEL
LIN {X 0,Y 351.086,Z 1002.531,A -85,B 0,C 180,E1 6476.533,E2 6476.533} C_VEL
LIN {X 0,Y 337.993,Z 1022.264,A -85,B 0,C 180,E1 6475.487,E2 6475.487} C_VEL
LIN {X 0,Y 326.464,Z 1038.153,A -85,B 0,C 180,E1 6474.474,E2 6474.474} C_VEL
LIN {X 0,Y 311.258,Z 1057.261,A -85,B 0,C 180,E1 6473.016,E2 6473.016} C_VEL
LIN {X 0,Y 295.341,Z 1075.121,A -85,B 0,C 180,E1 6471.31,E2 6471.31} C_VEL
LIN {X 0,Y 276.993,Z 1093.67,A -85,B 0,C 180,E1 6469.054,E2 6469.054} C_VEL
LIN {X 0,Y 260.881,Z 1108.46,A -85,B 0,C 180,E1 6466.769,E2 6466.769} C_VEL
LIN {X 0,Y 242.648,Z 1123.616,A -85,B 0,C 180,E1 6463.753,E2 6463.753} C_VEL
LIN {X 0,Y 227.178,Z 1135.456,A -85,B 0,C 180,E1 6460.725,E2 6460.725} C_VEL
LIN {X 0,Y 208.541,Z 1148.546,A -85,B 0,C 180,E1 6456.307,E2 6456.307} C_VEL
LIN {X 0,Y 191.602,Z 1159.567,A -85,B 0,C 180,E1 6451.24,E2 6451.24} C_VEL
LIN {X 0,Y 175.635,Z 1169.095,A -85,B 0,C 180,E1 6445.056,E2 6445.056} C_VEL
LIN {X 0,Y 160.841,Z 1177.608,A -85,B 0,C 180,E1 6437.179,E2 6437.179} C_VEL
LIN {X 0,Y 149.6,Z 1184.119,A -85,B 0,C 180,E1 6428.425,E2 6428.425} C_VEL
LIN {X 0,Y 141.716,Z 1188.89,A -85,B 0,C 180,E1 6418.665,E2 6418.665} C_VEL
LIN {X 0,Y 137.259,Z 1192.312,A -85,B 0,C 180,E1 6407.81,E2 6407.81} C_VEL
LIN {X 0,Y 136.125,Z 1193.834,A -85,B 0,C 180,E1 6399.294,E2 6399.294} C_VEL
LIN {X 0,Y 136.058,Z 1194.378,A -85,B 0,C 180,E1 6392.522,E2 6392.522} C_VEL
LIN {X 0,Y 136.049,Z 1194.338,A -85,B 0,C 180,E1 6386.624,E2 6386.624} C_VEL
LIN {X 0,Y 136.191,Z 1193.661,A -85,B 0,C 180,E1 6379.419,E2 6379.419} C_VEL
LIN {X 0,Y 137.965,Z 1191.683,A -85,B 0,C 180,E1 6369.637,E2 6369.637} C_VEL
LIN {X 0,Y 142.749,Z 1188.202,A -85,B 0,C 180,E1 6359.708,E2 6359.708} C_VEL
LIN {X 0,Y 152.009,Z 1182.611,A -85,B 0,C 180,E1 6349.362,E2 6349.362} C_VEL
LIN {X 0,Y 164.554,Z 1175.486,A -85,B 0,C 180,E1 6340.57,E2 6340.57} C_VEL
LIN {X 0,Y 179.452,Z 1166.814,A -85,B 0,C 180,E1 6333.296,E2 6333.296} C_VEL
LIN {X 0,Y 196.608,Z 1156.258,A -85,B 0,C 180,E1 6327.121,E2 6327.121} C_VEL
LIN {X 0,Y 214.301,Z 1144.54,A -85,B 0,C 180,E1 6322.17,E2 6322.17} C_VEL
LIN {X 0,Y 195.221,Z 1149.781,A -85,B 0,C 180,E1 6317.897,E2 6317.897} C_VEL
LIN {X 0,Y 178.442,Z 1153.937,A -85,B 0,C 180,E1 6312.294,E2 6312.294} C_VEL
LIN {X 0,Y 164.972,Z 1157.208,A -85,B 0,C 180,E1 6305.216,E2 6305.216} C_VEL
LIN {X 0,Y 154.879,Z 1160.007,A -85,B 0,C 180,E1 6295.557,E2 6295.557} C_VEL
LIN {X 0,Y 150.945,Z 1162.459,A -85,B 0,C 180,E1 6283.054,E2 6283.054} C_VEL
LIN {X 0,Y 157.709,Z 1164.48,A -85,B 0,C 180,E1 6268.249,E2 6268.249} C_VEL
LIN {X 0,Y 167.907,Z 1165.344,A -85,B 0,C 180,E1 6259.932,E2 6259.932} C_VEL
LIN {X 0,Y 155.971,Z 1172.137,A -85,B 0,C 180,E1 6252.314,E2 6252.314} C_VEL
LIN {X 0,Y 145.586,Z 1178.196,A -85,B 0,C 180,E1 6242.352,E2 6242.352} C_VEL
LIN {X 0,Y 139.894,Z 1181.878,A -85,B 0,C 180,E1 6233.153,E2 6233.153} C_VEL
LIN {X 0,Y 136.873,Z 1184.365,A -85,B 0,C 180,E1 6223.094,E2 6223.094} C_VEL
LIN {X 0,Y 136.139,Z 1185.307,A -85,B 0,C 180,E1 6215.061,E2 6215.061} C_VEL
LIN {X 0,Y 136.08,Z 1185.474,A -85,B 0,C 180,E1 6208.321,E2 6208.321} C_VEL
LIN {X 0,Y 136.388,Z 1184.927,A -85,B 0,C 180,E1 6200.724,E2 6200.724} C_VEL
LIN {X 0,Y 137.878,Z 1183.414,A -85,B 0,C 180,E1 6192.273,E2 6192.273} C_VEL
LIN {X 0,Y 141.737,Z 1180.668,A -85,B 0,C 180,E1 6183.167,E2 6183.167} C_VEL
LIN {X 0,Y 149.68,Z 1175.807,A -85,B 0,C 180,E1 6173.049,E2 6173.049} C_VEL
LIN {X 0,Y 160.153,Z 1169.838,A -85,B 0,C 180,E1 6164.63,E2 6164.63} C_VEL
LIN {X 0,Y 173.898,Z 1161.905,A -85,B 0,C 180,E1 6156.951,E2 6156.951} C_VEL
LIN {X 0,Y 189.421,Z 1152.794,A -85,B 0,C 180,E1 6150.645,E2 6150.645} C_VEL
LIN {X 0,Y 206.717,Z 1141.754,A -85,B 0,C 180,E1 6145.252,E2 6145.252} C_VEL
LIN {X 0,Y 224.728,Z 1129.52,A -85,B 0,C 180,E1 6140.852,E2 6140.852} C_VEL
LIN {X 0,Y 241.185,Z 1117.305,A -85,B 0,C 180,E1 6137.55,E2 6137.55} C_VEL
LIN {X 0,Y 259.227,Z 1102.811,A -85,B 0,C 180,E1 6134.512,E2 6134.512} C_VEL
LIN {X 0,Y 276.08,Z 1087.99,A -85,B 0,C 180,E1 6132.093,E2 6132.093} C_VEL
LIN {X 0,Y 294.273,Z 1070.279,A -85,B 0,C 180,E1 6129.832,E2 6129.832} C_VEL
LIN {X 0,Y 310.984,Z 1052.315,A -85,B 0,C 180,E1 6128.012,E2 6128.012} C_VEL
LIN {X 0,Y 326.29,Z 1033.787,A -85,B 0,C 180,E1 6126.51,E2 6126.51} C_VEL
LIN {X 0,Y 341.335,Z 1013.578,A -85,B 0,C 180,E1 6125.173,E2 6125.173} C_VEL
LIN {X 0,Y 352.897,Z 996.164,A -85,B 0,C 180,E1 6124.214,E2 6124.214} C_VEL
LIN {X 0,Y 365.52,Z 974.744,A -85,B 0,C 180,E1 6123.223,E2 6123.223} C_VEL
LIN {X 0,Y 375.297,Z 955.975,A -85,B 0,C 180,E1 6122.498,E2 6122.498} C_VEL
LIN {X 0,Y 385.126,Z 934.089,A -85,B 0,C 180,E1 6121.785,E2 6121.785} C_VEL
LIN {X 0,Y 393.275,Z 913.034,A -85,B 0,C 180,E1 6121.204,E2 6121.204} C_VEL
LIN {X 0,Y 406.569,Z 873.201,A -85,B 0,C 180,E1 6120.348,E2 6120.348} C_VEL
LIN {X 0,Y 407.658,Z 869.782,A -85,B 0,C 180,E1 6120.263,E2 6120.263} C_VEL
LIN {X 0,Y 407.237,Z 871.192,A -85,B 0,C 180,E1 6120.177,E2 6120.177} C_VEL
LIN {X 0,Y 393.955,Z 911.821,A -85,B 0,C 180,E1 6119.463,E2 6119.463} C_VEL
LIN {X 0,Y 385.009,Z 935.62,A -85,B 0,C 180,E1 6118.91,E2 6118.91} C_VEL
LIN {X 0,Y 375.113,Z 958.352,A -85,B 0,C 180,E1 6118.26,E2 6118.26} C_VEL
LIN {X 0,Y 364.283,Z 979.484,A -85,B 0,C 180,E1 6117.519,E2 6117.519} C_VEL
LIN {X 0,Y 363.273,Z 981.361,A -85,B 0,C 180,E1 6117.447,E2 6117.447} C_VEL
LIN {X 0,Y 359.462,Z 988.264,A -85,B 0,C 180,E1 6117.336,E2 6117.336} C_VEL
LIN {X 0,Y 348.62,Z 1005.082,A -85,B 0,C 180,E1 6117.568,E2 6117.568} C_VEL
LIN {X 0,Y 344.423,Z 1011.432,A -85,B 0,C 180,E1 6117.425,E2 6117.425} C_VEL
LIN {X 0,Y 329.645,Z 1032.367,A -85,B 0,C 180,E1 6116.268,E2 6116.268} C_VEL
LIN {X 0,Y 317.442,Z 1047.967,A -85,B 0,C 180,E1 6115.216,E2 6115.216} C_VEL
LIN {X 0,Y 302.717,Z 1065.351,A -85,B 0,C 180,E1 6113.806,E2 6113.806} C_VEL
LIN {X 0,Y 285.738,Z 1083.144,A -85,B 0,C 180,E1 6111.992,E2 6111.992} C_VEL
LIN {X 0,Y 268.168,Z 1099.971,A -85,B 0,C 180,E1 6109.83,E2 6109.83} C_VEL
LIN {X 0,Y 250.118,Z 1115.384,A -85,B 0,C 180,E1 6107.257,E2 6107.257} C_VEL
LIN {X 0,Y 231.769,Z 1129.736,A -85,B 0,C 180,E1 6104.152,E2 6104.152} C_VEL
LIN {X 0,Y 214.977,Z 1141.602,A -85,B 0,C 180,E1 6100.754,E2 6100.754} C_VEL
LIN {X 0,Y 197.46,Z 1153.127,A -85,B 0,C 180,E1 6096.414,E2 6096.414} C_VEL
LIN {X 0,Y 180.463,Z 1163.298,A -85,B 0,C 180,E1 6091.086,E2 6091.086} C_VEL
LIN {X 0,Y 163.832,Z 1172.63,A -85,B 0,C 180,E1 6084.133,E2 6084.133} C_VEL
LIN {X 0,Y 150.023,Z 1180.11,A -85,B 0,C 180,E1 6076.031,E2 6076.031} C_VEL
LIN {X 0,Y 139.033,Z 1185.983,A -85,B 0,C 180,E1 6066.343,E2 6066.343} C_VEL
LIN {X 0,Y 131.852,Z 1190.271,A -85,B 0,C 180,E1 6055.52,E2 6055.52} C_VEL
LIN {X 0,Y 128.778,Z 1192.704,A -85,B 0,C 180,E1 6045.677,E2 6045.677} C_VEL
LIN {X 0,Y 128.06,Z 1193.936,A -85,B 0,C 180,E1 6036.72,E2 6036.72} C_VEL
LIN {X 0,Y 128.075,Z 1194.202,A -85,B 0,C 180,E1 6029.547,E2 6029.547} C_VEL
LIN {X 0,Y 128.078,Z 1193.839,A -85,B 0,C 180,E1 6022.368,E2 6022.368} C_VEL
LIN {X 0,Y 129.064,Z 1192.397,A -85,B 0,C 180,E1 6012.873,E2 6012.873} C_VEL
LIN {X 0,Y 132.987,Z 1189.567,A -85,B 0,C 180,E1 6002.209,E2 6002.209} C_VEL
LIN {X 0,Y 141.132,Z 1184.806,A -85,B 0,C 180,E1 5991.425,E2 5991.425} C_VEL
LIN {X 0,Y 153.639,Z 1178.081,A -85,B 0,C 180,E1 5981.54,E2 5981.54} C_VEL
LIN {X 0,Y 169.001,Z 1169.756,A -85,B 0,C 180,E1 5973.459,E2 5973.459} C_VEL
LIN {X 0,Y 186.224,Z 1159.908,A -85,B 0,C 180,E1 5966.956,E2 5966.956} C_VEL
LIN {X 0,Y 202.17,Z 1150.004,A -85,B 0,C 180,E1 5962.271,E2 5962.271} C_VEL
LIN {X 0,Y 183.625,Z 1154.546,A -85,B 0,C 180,E1 5957.64,E2 5957.64} C_VEL
LIN {X 0,Y 167.869,Z 1158.075,A -85,B 0,C 180,E1 5951.684,E2 5951.684} C_VEL
LIN {X 0,Y 156.571,Z 1160.608,A -85,B 0,C 180,E1 5945.129,E2 5945.129} C_VEL
LIN {X 0,Y 147.043,Z 1163.025,A -85,B 0,C 180,E1 5935.319,E2 5935.319} C_VEL
LIN {X 0,Y 143.403,Z 1165.138,A -85,B 0,C 180,E1 5922.807,E2 5922.807} C_VEL
LIN {X 0,Y 150.192,Z 1166.974,A -85,B 0,C 180,E1 5907.732,E2 5907.732} C_VEL
LIN {X 0,Y 158.898,Z 1167.684,A -85,B 0,C 180,E1 5900.154,E2 5900.154} C_VEL
LIN {X 0,Y 145.323,Z 1174.91,A -85,B 0,C 180,E1 5890.812,E2 5890.812} C_VEL
LIN {X 0,Y 136.778,Z 1179.561,A -85,B 0,C 180,E1 5881.764,E2 5881.764} C_VEL
LIN {X 0,Y 130.764,Z 1183.248,A -85,B 0,C 180,E1 5870.599,E2 5870.599} C_VEL
LIN {X 0,Y 128.653,Z 1184.932,A -85,B 0,C 180,E1 5861.664,E2 5861.664} C_VEL
LIN {X 0,Y 128.113,Z 1185.629,A -85,B 0,C 180,E1 5854.033,E2 5854.033} C_VEL
LIN {X 0,Y 128.089,Z 1185.696,A -85,B 0,C 180,E1 5847.321,E2 5847.321} C_VEL
LIN {X 0,Y 128.494,Z 1185.133,A -85,B 0,C 180,E1 5839.696,E2 5839.696} C_VEL
LIN {X 0,Y 130.293,Z 1183.583,A -85,B 0,C 180,E1 5830.723,E2 5830.723} C_VEL
LIN {X 0,Y 135.263,Z 1180.532,A -85,B 0,C 180,E1 5820.319,E2 5820.319} C_VEL
LIN {X 0,Y 143.966,Z 1175.652,A -85,B 0,C 180,E1 5810.292,E2 5810.292} C_VEL
LIN {X 0,Y 156.041,Z 1169.338,A -85,B 0,C 180,E1 5801.442,E2 5801.442} C_VEL
LIN {X 0,Y 170.956,Z 1161.216,A -85,B 0,C 180,E1 5793.855,E2 5793.855} C_VEL
LIN {X 0,Y 188.914,Z 1150.952,A -85,B 0,C 180,E1 5787.238,E2 5787.238} C_VEL
LIN {X 0,Y 207.257,Z 1139.752,A -85,B 0,C 180,E1 5782.149,E2 5782.149} C_VEL
LIN {X 0,Y 224.363,Z 1128.172,A -85,B 0,C 180,E1 5778.345,E2 5778.345} C_VEL
LIN {X 0,Y 242.353,Z 1115.234,A -85,B 0,C 180,E1 5775.066,E2 5775.066} C_VEL
LIN {X 0,Y 260.871,Z 1100.328,A -85,B 0,C 180,E1 5772.225,E2 5772.225} C_VEL
LIN {X 0,Y 279.994,Z 1083.445,A -85,B 0,C 180,E1 5769.746,E2 5769.746} C_VEL
LIN {X 0,Y 295.799,Z 1067.971,A -85,B 0,C 180,E1 5767.957,E2 5767.957} C_VEL
LIN {X 0,Y 312.329,Z 1050.09,A -85,B 0,C 180,E1 5766.29,E2 5766.29} C_VEL
LIN {X 0,Y 328.129,Z 1031.215,A -85,B 0,C 180,E1 5764.866,E2 5764.866} C_VEL
LIN {X 0,Y 343.129,Z 1010.731,A -85,B 0,C 180,E1 5763.62,E2 5763.62} C_VEL
LIN {X 0,Y 356.314,Z 990.537,A -85,B 0,C 180,E1 5762.615,E2 5762.615} C_VEL
LIN {X 0,Y 367.128,Z 971.887,A -85,B 0,C 180,E1 5761.825,E2 5761.825} C_VEL
LIN {X 0,Y 378.501,Z 949.337,A -85,B 0,C 180,E1 5761.032,E2 5761.032} C_VEL
LIN {X 0,Y 387.948,Z 927.654,A -85,B 0,C 180,E1 5760.395,E2 5760.395} C_VEL
LIN {X 0,Y 388.651,Z 925.831,A -85,B 0,C 180,E1 5760.346,E2 5760.346} C_VEL
LIN {X 0,Y 378.657,Z 949.583,A -85,B 0,C 180,E1 5759.748,E2 5759.748} C_VEL
LIN {X 0,Y 367.543,Z 972.487,A -85,B 0,C 180,E1 5759.043,E2 5759.043} C_VEL
LIN {X 0,Y 355.117,Z 994.398,A -85,B 0,C 180,E1 5758.207,E2 5758.207} C_VEL
LIN {X 0,Y 344.423,Z 1011.432,A -85,B 0,C 180,E1 5757.425,E2 5757.425} C_VEL
LIN {X 0,Y 340.115,Z 1017.832,A -85,B 0,C 180,E1 5757.27,E2 5757.27} C_VEL
LIN {X 0,Y 327.928,Z 1033.822,A -85,B 0,C 180,E1 5757.423,E2 5757.423} C_VEL
LIN {X 0,Y 323.099,Z 1039.783,A -85,B 0,C 180,E1 5757.228,E2 5757.228} C_VEL
LIN {X 0,Y 308.208,Z 1057.489,A -85,B 0,C 180,E1 5755.977,E2 5755.977} C_VEL
LIN {X 0,Y 294.707,Z 1072.296,A -85,B 0,C 180,E1 5754.709,E2 5754.709} C_VEL
LIN {X 0,Y 277.112,Z 1089.879,A -85,B 0,C 180,E1 5752.843,E2 5752.843} C_VEL
LIN {X 0,Y 260.305,Z 1104.965,A -85,B 0,C 180,E1 5750.798,E2 5750.798} C_VEL
LIN {X 0,Y 240.256,Z 1121.239,A -85,B 0,C 180,E1 5747.946,E2 5747.946} C_VEL
LIN {X 0,Y 221.741,Z 1134.817,A -85,B 0,C 180,E1 5744.777,E2 5744.777} C_VEL
LIN {X 0,Y 203.142,Z 1147.075,A -85,B 0,C 180,E1 5740.904,E2 5740.904} C_VEL
LIN {X 0,Y 186.356,Z 1157.337,A -85,B 0,C 180,E1 5736.551,E2 5736.551} C_VEL
LIN {X 0,Y 168.629,Z 1167.198,A -85,B 0,C 180,E1 5730.64,E2 5730.64} C_VEL
LIN {X 0,Y 152.65,Z 1175.579,A -85,B 0,C 180,E1 5723.411,E2 5723.411} C_VEL
LIN {X 0,Y 138.754,Z 1182.494,A -85,B 0,C 180,E1 5714.339,E2 5714.339} C_VEL
LIN {X 0,Y 128.298,Z 1187.812,A -85,B 0,C 180,E1 5703.497,E2 5703.497} C_VEL
LIN {X 0,Y 122.36,Z 1191.374,A -85,B 0,C 180,E1 5692.073,E2 5692.073} C_VEL
LIN {X 0,Y 120.252,Z 1193.184,A -85,B 0,C 180,E1 5681.505,E2 5681.505} C_VEL
LIN {X 0,Y 120.053,Z 1193.812,A -85,B 0,C 180,E1 5673.815,E2 5673.815} C_VEL
LIN {X 0,Y 120.065,Z 1193.867,A -85,B 0,C 180,E1 5667.608,E2 5667.608} C_VEL
LIN {X 0,Y 120.161,Z 1193.347,A -85,B 0,C 180,E1 5659.93,E2 5659.93} C_VEL
LIN {X 0,Y 121.774,Z 1191.738,A -85,B 0,C 180,E1 5649.821,E2 5649.821} C_VEL
LIN {X 0,Y 127.429,Z 1188.274,A -85,B 0,C 180,E1 5637.747,E2 5637.747} C_VEL
LIN {X 0,Y 137.359,Z 1183.189,A -85,B 0,C 180,E1 5626.816,E2 5626.816} C_VEL
LIN {X 0,Y 151.111,Z 1176.275,A -85,B 0,C 180,E1 5617.43,E2 5617.43} C_VEL
LIN {X 0,Y 167.98,Z 1167.509,A -85,B 0,C 180,E1 5609.607,E2 5609.607} C_VEL
LIN {X 0,Y 187.144,Z 1156.799,A -85,B 0,C 180,E1 5603.216,E2 5603.216} C_VEL
LIN {X 0,Y 190.089,Z 1155.035,A -85,B 0,C 180,E1 5602.337,E2 5602.337} C_VEL
LIN {X 0,Y 172.784,Z 1158.772,A -85,B 0,C 180,E1 5597.513,E2 5597.513} C_VEL
LIN {X 0,Y 156.665,Z 1162.082,A -85,B 0,C 180,E1 5590.666,E2 5590.666} C_VEL
LIN {X 0,Y 142.675,Z 1165.025,A -85,B 0,C 180,E1 5580,E2 5580} C_VEL
LIN {X 0,Y 136.07,Z 1167.248,A -85,B 0,C 180,E1 5566.4,E2 5566.4} C_VEL
LIN {X 0,Y 139.578,Z 1168.963,A -85,B 0,C 180,E1 5551.317,E2 5551.317} C_VEL
LIN {X 0,Y 149.919,Z 1169.982,A -85,B 0,C 180,E1 5540.413,E2 5540.413} C_VEL
LIN {X 0,Y 136.878,Z 1176.327,A -85,B 0,C 180,E1 5531.111,E2 5531.111} C_VEL
LIN {X 0,Y 127.338,Z 1181.184,A -85,B 0,C 180,E1 5520.174,E2 5520.174} C_VEL
LIN {X 0,Y 122.492,Z 1183.918,A -85,B 0,C 180,E1 5510.056,E2 5510.056} C_VEL
LIN {X 0,Y 120.522,Z 1185.432,A -85,B 0,C 180,E1 5500.522,E2 5500.522} C_VEL
LIN {X 0,Y 120.092,Z 1185.971,A -85,B 0,C 180,E1 5492.392,E2 5492.392} C_VEL
LIN {X 0,Y 120.135,Z 1185.882,A -85,B 0,C 180,E1 5485.232,E2 5485.232} C_VEL
LIN {X 0,Y 120.804,Z 1185.164,A -85,B 0,C 180,E1 5477.093,E2 5477.093} C_VEL
LIN {X 0,Y 123.877,Z 1183.171,A -85,B 0,C 180,E1 5466.204,E2 5466.204} C_VEL
LIN {X 0,Y 130.467,Z 1179.554,A -85,B 0,C 180,E1 5455.457,E2 5455.457} C_VEL
LIN {X 0,Y 140.517,Z 1174.638,A -85,B 0,C 180,E1 5445.793,E2 5445.793} C_VEL
LIN {X 0,Y 154.314,Z 1167.765,A -85,B 0,C 180,E1 5437.057,E2 5437.057} C_VEL
LIN {X 0,Y 170.6,Z 1159.444,A -85,B 0,C 180,E1 5429.849,E2 5429.849} C_VEL
LIN {X 0,Y 187.55,Z 1149.984,A -85,B 0,C 180,E1 5424.276,E2 5424.276} C_VEL
LIN {X 0,Y 205.907,Z 1139.087,A -85,B 0,C 180,E1 5419.611,E2 5419.611} C_VEL
LIN {X 0,Y 223.612,Z 1127.483,A -85,B 0,C 180,E1 5415.99,E2 5415.99} C_VEL
LIN {X 0,Y 244.435,Z 1112.515,A -85,B 0,C 180,E1 5412.521,E2 5412.521} C_VEL
LIN {X 0,Y 263.843,Z 1097.106,A -85,B 0,C 180,E1 5409.849,E2 5409.849} C_VEL
LIN {X 0,Y 281.588,Z 1081.278,A -85,B 0,C 180,E1 5407.755,E2 5407.755} C_VEL
LIN {X 0,Y 299.543,Z 1063.656,A -85,B 0,C 180,E1 5405.912,E2 5405.912} C_VEL
LIN {X 0,Y 314.922,Z 1046.882,A -85,B 0,C 180,E1 5404.506,E2 5404.506} C_VEL
LIN {X 0,Y 329.846,Z 1028.709,A -85,B 0,C 180,E1 5403.259,E2 5403.259} C_VEL
LIN {X 0,Y 343.698,Z 1010.071,A -85,B 0,C 180,E1 5402.201,E2 5402.201} C_VEL
LIN {X 0,Y 357.028,Z 989.599,A -85,B 0,C 180,E1 5401.25,E2 5401.25} C_VEL
LIN {X 0,Y 369.136,Z 968.626,A -85,B 0,C 180,E1 5400.429,E2 5400.429} C_VEL
LIN {X 0,Y 356.45,Z 991.265,A -85,B 0,C 180,E1 5399.64,E2 5399.64} C_VEL
LIN {X 0,Y 342.484,Z 1013.328,A -85,B 0,C 180,E1 5398.687,E2 5398.687} C_VEL
LIN {X 0,Y 328.224,Z 1032.986,A -85,B 0,C 180,E1 5397.643,E2 5397.643} C_VEL
LIN {X 0,Y 323.099,Z 1039.783,A -85,B 0,C 180,E1 5397.228,E2 5397.228} C_VEL
LIN {X 0,Y 318.171,Z 1045.671,A -85,B 0,C 180,E1 5397.017,E2 5397.017} C_VEL
LIN {X 0,Y 303.907,Z 1061.417,A -85,B 0,C 180,E1 5397.051,E2 5397.051} C_VEL
LIN {X 0,Y 299.382,Z 1066.095,A -85,B 0,C 180,E1 5396.815,E2 5396.815} C_VEL
LIN {X 0,Y 285.325,Z 1080.44,A -85,B 0,C 180,E1 5395.516,E2 5395.516} C_VEL
LIN {X 0,Y 270.451,Z 1094.485,A -85,B 0,C 180,E1 5393.968,E2 5393.968} C_VEL
LIN {X 0,Y 250.65,Z 1111.339,A -85,B 0,C 180,E1 5391.593,E2 5391.593} C_VEL
LIN {X 0,Y 231.333,Z 1126.174,A -85,B 0,C 180,E1 5388.841,E2 5388.841} C_VEL
LIN {X 0,Y 211.737,Z 1139.558,A -85,B 0,C 180,E1 5385.466,E2 5385.466} C_VEL
LIN {X 0,Y 192.137,Z 1151.753,A -85,B 0,C 180,E1 5381.273,E2 5381.273} C_VEL
LIN {X 0,Y 174.469,Z 1161.635,A -85,B 0,C 180,E1 5376.475,E2 5376.475} C_VEL
LIN {X 0,Y 156.074,Z 1171.142,A -85,B 0,C 180,E1 5369.858,E2 5369.858} C_VEL
LIN {X 0,Y 140.635,Z 1178.58,A -85,B 0,C 180,E1 5362.1,E2 5362.1} C_VEL
LIN {X 0,Y 127.572,Z 1184.619,A -85,B 0,C 180,E1 5352.373,E2 5352.373} C_VEL
LIN {X 0,Y 118.018,Z 1189.266,A -85,B 0,C 180,E1 5340.546,E2 5340.546} C_VEL
LIN {X 0,Y 113.41,Z 1191.945,A -85,B 0,C 180,E1 5329.032,E2 5329.032} C_VEL
LIN {X 0,Y 112.091,Z 1193.386,A -85,B 0,C 180,E1 5318.044,E2 5318.044} C_VEL
LIN {X 0,Y 112.088,Z 1193.692,A -85,B 0,C 180,E1 5309.994,E2 5309.994} C_VEL
LIN {X 0,Y 112.091,Z 1193.379,A -85,B 0,C 180,E1 5301.958,E2 5301.958} C_VEL
LIN {X 0,Y 113.413,Z 1191.936,A -85,B 0,C 180,E1 5290.955,E2 5290.955} C_VEL
LIN {X 0,Y 118.311,Z 1189.11,A -85,B 0,C 180,E1 5278.96,E2 5278.96} C_VEL
LIN {X 0,Y 128.037,Z 1184.366,A -85,B 0,C 180,E1 5267.195,E2 5267.195} C_VEL
LIN {X 0,Y 142.438,Z 1177.668,A -85,B 0,C 180,E1 5256.838,E2 5256.838} C_VEL
LIN {X 0,Y 158.887,Z 1169.743,A -85,B 0,C 180,E1 5248.978,E2 5248.978} C_VEL
LIN {X 0,Y 178.217,Z 1159.569,A -85,B 0,C 180,E1 5242.384,E2 5242.384} C_VEL
LIN {X 0,Y 160.19,Z 1163.062,A -85,B 0,C 180,E1 5236.686,E2 5236.686} C_VEL
LIN {X 0,Y 145.164,Z 1165.794,A -85,B 0,C 180,E1 5229.115,E2 5229.115} C_VEL
LIN {X 0,Y 133.033,Z 1168.13,A -85,B 0,C 180,E1 5217.846,E2 5217.846} C_VEL
LIN {X 0,Y 128.201,Z 1170.039,A -85,B 0,C 180,E1 5203.619,E2 5203.619} C_VEL
LIN {X 0,Y 135.225,Z 1171.64,A -85,B 0,C 180,E1 5186.319,E2 5186.319} C_VEL
LIN {X 0,Y 140.861,Z 1172.037,A -85,B 0,C 180,E1 5180.697,E2 5180.697} C_VEL
LIN {X 0,Y 127.551,Z 1178.165,A -85,B 0,C 180,E1 5170.597,E2 5170.597} C_VEL
LIN {X 0,Y 118.502,Z 1182.307,A -85,B 0,C 180,E1 5159.307,E2 5159.307} C_VEL
LIN {X 0,Y 113.799,Z 1184.882,A -85,B 0,C 180,E1 5147.916,E2 5147.916} C_VEL
LIN {X 0,Y 112.247,Z 1186.065,A -85,B 0,C 180,E1 5137.17,E2 5137.17} C_VEL
LIN {X 0,Y 112.088,Z 1186.302,A -85,B 0,C 180,E1 5128.984,E2 5128.984} C_VEL
LIN {X 0,Y 112.427,Z 1185.9,A -85,B 0,C 180,E1 5120.278,E2 5120.278} C_VEL
LIN {X 0,Y 114.506,Z 1184.424,A -85,B 0,C 180,E1 5109.563,E2 5109.563} C_VEL
LIN {X 0,Y 119.317,Z 1181.938,A -85,B 0,C 180,E1 5099.264,E2 5099.264} C_VEL
LIN {X 0,Y 129.262,Z 1177.374,A -85,B 0,C 180,E1 5087.711,E2 5087.711} C_VEL
LIN {X 0,Y 141.351,Z 1171.861,A -85,B 0,C 180,E1 5078.92,E2 5078.92} C_VEL
LIN {X 0,Y 158.029,Z 1163.989,A -85,B 0,C 180,E1 5070.637,E2 5070.637} C_VEL
LIN {X 0,Y 174.88,Z 1155.487,A -85,B 0,C 180,E1 5064.631,E2 5064.631} C_VEL
LIN {X 0,Y 193.211,Z 1145.35,A -85,B 0,C 180,E1 5059.645,E2 5059.645} C_VEL
LIN {X 0,Y 211.843,Z 1134.226,A -85,B 0,C 180,E1 5055.677,E2 5055.677} C_VEL
LIN {X 0,Y 232.185,Z 1120.642,A -85,B 0,C 180,E1 5052.18,E2 5052.18} C_VEL
LIN {X 0,Y 253.231,Z 1105.041,A -85,B 0,C 180,E1 5049.225,E2 5049.225} C_VEL
LIN {X 0,Y 271.991,Z 1089.613,A -85,B 0,C 180,E1 5047.016,E2 5047.016} C_VEL
LIN {X 0,Y 289.164,Z 1073.751,A -85,B 0,C 180,E1 5045.248,E2 5045.248} C_VEL
LIN {X 0,Y 305.736,Z 1057.12,A -85,B 0,C 180,E1 5043.75,E2 5043.75} C_VEL
LIN {X 0,Y 322.722,Z 1037.742,A -85,B 0,C 180,E1 5042.366,E2 5042.366} C_VEL
LIN {X 0,Y 338.772,Z 1017.18,A -85,B 0,C 180,E1 5041.184,E2 5041.184} C_VEL
LIN {X 0,Y 348.731,Z 1003.019,A -85,B 0,C 180,E1 5040.493,E2 5040.493} C_VEL
LIN {X 0,Y 333.958,Z 1024.561,A -85,B 0,C 180,E1 5039.515,E2 5039.515} C_VEL
LIN {X 0,Y 318.401,Z 1044.403,A -85,B 0,C 180,E1 5038.38,E2 5038.38} C_VEL
LIN {X 0,Y 302.345,Z 1063.032,A -85,B 0,C 180,E1 5037.07,E2 5037.07} C_VEL
LIN {X 0,Y 299.382,Z 1066.095,A -85,B 0,C 180,E1 5036.815,E2 5036.815} C_VEL
LIN {X 0,Y 293.979,Z 1071.677,A -85,B 0,C 180,E1 5036.542,E2 5036.542} C_VEL
LIN {X 0,Y 278.446,Z 1086.132,A -85,B 0,C 180,E1 5036.442,E2 5036.442} C_VEL
LIN {X 0,Y 273.643,Z 1090.315,A -85,B 0,C 180,E1 5036.146,E2 5036.146} C_VEL
LIN {X 0,Y 258.14,Z 1103.835,A -85,B 0,C 180,E1 5034.508,E2 5034.508} C_VEL
LIN {X 0,Y 237.893,Z 1119.732,A -85,B 0,C 180,E1 5032.027,E2 5032.027} C_VEL
LIN {X 0,Y 220.64,Z 1131.963,A -85,B 0,C 180,E1 5029.521,E2 5029.521} C_VEL
LIN {X 0,Y 199.502,Z 1145.464,A -85,B 0,C 180,E1 5025.784,E2 5025.784} C_VEL
LIN {X 0,Y 179.456,Z 1156.998,A -85,B 0,C 180,E1 5021.284,E2 5021.284} C_VEL
LIN {X 0,Y 160.521,Z 1166.651,A -85,B 0,C 180,E1 5015.725,E2 5015.725} C_VEL
LIN {X 0,Y 142.838,Z 1175.022,A -85,B 0,C 180,E1 5008.641,E2 5008.641} C_VEL
LIN {X 0,Y 127.867,Z 1181.575,A -85,B 0,C 180,E1 5000.017,E2 5000.017} C_VEL
LIN {X 0,Y 115.263,Z 1187.014,A -85,B 0,C 180,E1 4988.644,E2 4988.644} C_VEL
LIN {X 0,Y 107.502,Z 1190.707,A -85,B 0,C 180,E1 4975.915,E2 4975.915} C_VEL
LIN {X 0,Y 104.458,Z 1192.581,A -85,B 0,C 180,E1 4963.838,E2 4963.838} C_VEL
LIN {X 0,Y 104.057,Z 1193.263,A -85,B 0,C 180,E1 4954.954,E2 4954.954} C_VEL
LIN {X 0,Y 104.074,Z 1193.356,A -85,B 0,C 180,E1 4947.681,E2 4947.681} C_VEL
LIN {X 0,Y 104.216,Z 1192.869,A -85,B 0,C 180,E1 4938.93,E2 4938.93} C_VEL
LIN {X 0,Y 106.344,Z 1191.273,A -85,B 0,C 180,E1 4927.319,E2 4927.319} C_VEL
LIN {X 0,Y 113.359,Z 1187.842,A -85,B 0,C 180,E1 4913.767,E2 4913.767} C_VEL
LIN {X 0,Y 125.135,Z 1182.775,A -85,B 0,C 180,E1 4901.995,E2 4901.995} C_VEL
LIN {X 0,Y 140.836,Z 1175.883,A -85,B 0,C 180,E1 4892.335,E2 4892.335} C_VEL
LIN {X 0,Y 160.263,Z 1166.779,A -85,B 0,C 180,E1 4884.361,E2 4884.361} C_VEL
LIN {X 0,Y 166.26,Z 1163.784,A -85,B 0,C 180,E1 4882.384,E2 4882.384} C_VEL
LIN {X 0,Y 147.868,Z 1166.9,A -85,B 0,C 180,E1 4875.693,E2 4875.693} C_VEL
LIN {X 0,Y 132.832,Z 1169.331,A -85,B 0,C 180,E1 4866.431,E2 4866.431} C_VEL
LIN {X 0,Y 121.881,Z 1171.544,A -85,B 0,C 180,E1 4851.508,E2 4851.508} C_VEL
LIN {X 0,Y 122.364,Z 1173.119,A -85,B 0,C 180,E1 4834.336,E2 4834.336} C_VEL
LIN {X 0,Y 131.82,Z 1174.068,A -85,B 0,C 180,E1 4821.038,E2 4821.038} C_VEL
LIN {X 0,Y 118.169,Z 1179.724,A -85,B 0,C 180,E1 4810.028,E2 4810.028} C_VEL
LIN {X 0,Y 109.666,Z 1183.413,A -85,B 0,C 180,E1 4798.308,E2 4798.308} C_VEL
LIN {X 0,Y 105.203,Z 1185.625,A -85,B 0,C 180,E1 4785.44,E2 4785.44} C_VEL
LIN {X 0,Y 104.19,Z 1186.385,A -85,B 0,C 180,E1 4776.066,E2 4776.066} C_VEL
LIN {X 0,Y 104.099,Z 1186.524,A -85,B 0,C 180,E1 4767.805,E2 4767.805} C_VEL
LIN {X 0,Y 104.614,Z 1186.046,A -85,B 0,C 180,E1 4758.428,E2 4758.428} C_VEL
LIN {X 0,Y 107.094,Z 1184.603,A -85,B 0,C 180,E1 4747.5,E2 4747.5} C_VEL
LIN {X 0,Y 113.366,Z 1181.816,A -85,B 0,C 180,E1 4735.642,E2 4735.642} C_VEL
LIN {X 0,Y 124.277,Z 1177.23,A -85,B 0,C 180,E1 4724.279,E2 4724.279} C_VEL
LIN {X 0,Y 138.172,Z 1171.409,A -85,B 0,C 180,E1 4715.152,E2 4715.152} C_VEL
LIN {X 0,Y 154.686,Z 1163.971,A -85,B 0,C 180,E1 4707.69,E2 4707.69} C_VEL
LIN {X 0,Y 173.175,Z 1155.11,A -85,B 0,C 180,E1 4701.642,E2 4701.642} C_VEL
LIN {X 0,Y 193.143,Z 1144.348,A -85,B 0,C 180,E1 4696.734,E2 4696.734} C_VEL
LIN {X 0,Y 214.62,Z 1131.591,A -85,B 0,C 180,E1 4692.648,E2 4692.648} C_VEL
LIN {X 0,Y 235.2,Z 1117.995,A -85,B 0,C 180,E1 4689.524,E2 4689.524} C_VEL
LIN {X 0,Y 253.93,Z 1104.027,A -85,B 0,C 180,E1 4687.149,E2 4687.149} C_VEL
LIN {X 0,Y 272.073,Z 1089.34,A -85,B 0,C 180,E1 4685.199,E2 4685.199} C_VEL
LIN {X 0,Y 289.293,Z 1073.617,A -85,B 0,C 180,E1 4683.567,E2 4683.567} C_VEL
LIN {X 0,Y 306.658,Z 1056.167,A -85,B 0,C 180,E1 4682.114,E2 4682.114} C_VEL
LIN {X 0,Y 322.489,Z 1038.405,A -85,B 0,C 180,E1 4680.927,E2 4680.927} C_VEL
LIN {X 0,Y 327.808,Z 1031.935,A -85,B 0,C 180,E1 4680.546,E2 4680.546} C_VEL
LIN {X 0,Y 309.973,Z 1053.485,A -85,B 0,C 180,E1 4679.284,E2 4679.284} C_VEL
LIN {X 0,Y 293.415,Z 1071.376,A -85,B 0,C 180,E1 4677.956,E2 4677.956} C_VEL
LIN {X 0,Y 275.519,Z 1088.626,A -85,B 0,C 180,E1 4676.328,E2 4676.328} C_VEL
LIN {X 0,Y 273.643,Z 1090.315,A -85,B 0,C 180,E1 4676.146,E2 4676.146} C_VEL
LIN {X 0,Y 267.913,Z 1095.446,A -85,B 0,C 180,E1 4675.8,E2 4675.8} C_VEL
LIN {X 0,Y 252.069,Z 1107.798,A -85,B 0,C 180,E1 4675.571,E2 4675.571} C_VEL
LIN {X 0,Y 246.097,Z 1112.287,A -85,B 0,C 180,E1 4675.157,E2 4675.157} C_VEL
LIN {X 0,Y 224.881,Z 1127.672,A -85,B 0,C 180,E1 4672.505,E2 4672.505} C_VEL
LIN {X 0,Y 207.209,Z 1139.174,A -85,B 0,C 180,E1 4669.843,E2 4669.843} C_VEL
LIN {X 0,Y 185.617,Z 1151.834,A -85,B 0,C 180,E1 4665.824,E2 4665.824} C_VEL
LIN {X 0,Y 165.1,Z 1162.581,A -85,B 0,C 180,E1 4660.854,E2 4660.854} C_VEL
LIN {X 0,Y 146.027,Z 1171.398,A -85,B 0,C 180,E1 4654.654,E2 4654.654} C_VEL
LIN {X 0,Y 128.983,Z 1178.731,A -85,B 0,C 180,E1 4646.837,E2 4646.837} C_VEL
LIN {X 0,Y 114.707,Z 1184.39,A -85,B 0,C 180,E1 4637.063,E2 4637.063} C_VEL
LIN {X 0,Y 103.067,Z 1189.083,A -85,B 0,C 180,E1 4623.563,E2 4623.563} C_VEL
LIN {X 0,Y 97.599,Z 1191.685,A -85,B 0,C 180,E1 4610.377,E2 4610.377} C_VEL
LIN {X 0,Y 96.092,Z 1192.914,A -85,B 0,C 180,E1 4597.767,E2 4597.767} C_VEL
LIN {X 0,Y 96.091,Z 1193.152,A -85,B 0,C 180,E1 4589.396,E2 4589.396} C_VEL
LIN {X 0,Y 96.14,Z 1192.83,A -85,B 0,C 180,E1 4580.414,E2 4580.414} C_VEL
LIN {X 0,Y 98.249,Z 1191.282,A -85,B 0,C 180,E1 4567.242,E2 4567.242} C_VEL
LIN {X 0,Y 105.202,Z 1188.235,A -85,B 0,C 180,E1 4553.209,E2 4553.209} C_VEL
LIN {X 0,Y 117.419,Z 1183.325,A -85,B 0,C 180,E1 4540.714,E2 4540.714} C_VEL
LIN {X 0,Y 134.412,Z 1176.417,A -85,B 0,C 180,E1 4530.345,E2 4530.345} C_VEL
LIN {X 0,Y 154.448,Z 1167.568,A -85,B 0,C 180,E1 4522.339,E2 4522.339} C_VEL
LIN {X 0,Y 135.085,Z 1170.416,A -85,B 0,C 180,E1 4514.138,E2 4514.138} C_VEL
LIN {X 0,Y 119.925,Z 1172.634,A -85,B 0,C 180,E1 4501.911,E2 4501.911} C_VEL
LIN {X 0,Y 113.05,Z 1174.293,A -85,B 0,C 180,E1 4486.184,E2 4486.184} C_VEL
LIN {X 0,Y 117.46,Z 1175.528,A -85,B 0,C 180,E1 4468.359,E2 4468.359} C_VEL
LIN {X 0,Y 122.766,Z 1175.942,A -85,B 0,C 180,E1 4461.442,E2 4461.442} C_VEL
LIN {X 0,Y 109.66,Z 1180.92,A -85,B 0,C 180,E1 4450.352,E2 4450.352} C_VEL
LIN {X 0,Y 100.525,Z 1184.478,A -85,B 0,C 180,E1 4436.465,E2 4436.465} C_VEL
LIN {X 0,Y 96.98,Z 1186.121,A -85,B 0,C 180,E1 4424.334,E2 4424.334} C_VEL
LIN {X 0,Y 96.146,Z 1186.703,A -85,B 0,C 180,E1 4414.78,E2 4414.78} C_VEL
LIN {X 0,Y 96.109,Z 1186.768,A -85,B 0,C 180,E1 4407.026,E2 4407.026} C_VEL
LIN {X 0,Y 96.79,Z 1186.258,A -85,B 0,C 180,E1 4396.871,E2 4396.871} C_VEL
LIN {X 0,Y 99.821,Z 1184.781,A -85,B 0,C 180,E1 4385.129,E2 4385.129} C_VEL
LIN {X 0,Y 107.472,Z 1181.836,A -85,B 0,C 180,E1 4372.126,E2 4372.126} C_VEL
LIN {X 0,Y 119.764,Z 1177.085,A -85,B 0,C 180,E1 4360.568,E2 4360.568} C_VEL
LIN {X 0,Y 135.611,Z 1170.925,A -85,B 0,C 180,E1 4351.219,E2 4351.219} C_VEL
LIN {X 0,Y 154.089,Z 1162.968,A -85,B 0,C 180,E1 4343.814,E2 4343.814} C_VEL
LIN {X 0,Y 175.331,Z 1152.901,A -85,B 0,C 180,E1 4337.769,E2 4337.769} C_VEL
LIN {X 0,Y 196.243,Z 1141.898,A -85,B 0,C 180,E1 4333.321,E2 4333.321} C_VEL
LIN {X 0,Y 216.224,Z 1129.969,A -85,B 0,C 180,E1 4329.967,E2 4329.967} C_VEL
LIN {X 0,Y 236.806,Z 1116.425,A -85,B 0,C 180,E1 4327.163,E2 4327.163} C_VEL
LIN {X 0,Y 255.925,Z 1102.388,A -85,B 0,C 180,E1 4324.989,E2 4324.989} C_VEL
LIN {X 0,Y 274.379,Z 1087.243,A -85,B 0,C 180,E1 4323.192,E2 4323.192} C_VEL
LIN {X 0,Y 292.079,Z 1071.298,A -85,B 0,C 180,E1 4321.696,E2 4321.696} C_VEL
LIN {X 0,Y 306.472,Z 1056.79,A -85,B 0,C 180,E1 4320.586,E2 4320.586} C_VEL
LIN {X 0,Y 287.484,Z 1076.432,A -85,B 0,C 180,E1 4319.144,E2 4319.144} C_VEL
LIN {X 0,Y 270.184,Z 1092.512,A -85,B 0,C 180,E1 4317.632,E2 4317.632} C_VEL
LIN {X 0,Y 250.582,Z 1108.78,A -85,B 0,C 180,E1 4315.652,E2 4315.652} C_VEL
LIN {X 0,Y 246.097,Z 1112.287,A -85,B 0,C 180,E1 4315.157,E2 4315.157} C_VEL
LIN {X 0,Y 240.033,Z 1116.802,A -85,B 0,C 180,E1 4314.714,E2 4314.714} C_VEL
LIN {X 0,Y 223.229,Z 1127.753,A -85,B 0,C 180,E1 4314.288,E2 4314.288} C_VEL
LIN {X 0,Y 216.98,Z 1131.824,A -85,B 0,C 180,E1 4313.743,E2 4313.743} C_VEL
LIN {X 0,Y 196.119,Z 1144.477,A -85,B 0,C 180,E1 4310.61,E2 4310.61} C_VEL
LIN {X 0,Y 175.649,Z 1155.711,A -85,B 0,C 180,E1 4306.74,E2 4306.74} C_VEL
LIN {X 0,Y 154.513,Z 1165.835,A -85,B 0,C 180,E1 4301.513,E2 4301.513} C_VEL
LIN {X 0,Y 133.323,Z 1174.886,A -85,B 0,C 180,E1 4294.14,E2 4294.14} C_VEL
LIN {X 0,Y 116.491,Z 1181.457,A -85,B 0,C 180,E1 4285.476,E2 4285.476} C_VEL
LIN {X 0,Y 102.291,Z 1186.564,A -85,B 0,C 180,E1 4273.939,E2 4273.939} C_VEL
LIN {X 0,Y 92.959,Z 1190.138,A -85,B 0,C 180,E1 4260.358,E2 4260.358} C_VEL
LIN {X 0,Y 88.745,Z 1192.04,A -85,B 0,C 180,E1 4246.352,E2 4246.352} C_VEL
LIN {X 0,Y 88.068,Z 1192.734,A -85,B 0,C 180,E1 4235.857,E2 4235.857} C_VEL
LIN {X 0,Y 88.084,Z 1192.852,A -85,B 0,C 180,E1 4228.04,E2 4228.04} C_VEL
LIN {X 0,Y 88.255,Z 1192.447,A -85,B 0,C 180,E1 4218.225,E2 4218.225} C_VEL
LIN {X 0,Y 90.951,Z 1190.911,A -85,B 0,C 180,E1 4204.603,E2 4204.603} C_VEL
LIN {X 0,Y 99.101,Z 1187.771,A -85,B 0,C 180,E1 4189.771,E2 4189.771} C_VEL
LIN {X 0,Y 112.744,Z 1182.779,A -85,B 0,C 180,E1 4177.034,E2 4177.034} C_VEL
LIN {X 0,Y 131.096,Z 1175.758,A -85,B 0,C 180,E1 4166.816,E2 4166.816} C_VEL
LIN {X 0,Y 142.54,Z 1170.984,A -85,B 0,C 180,E1 4162.177,E2 4162.177} C_VEL
LIN {X 0,Y 125.796,Z 1173.177,A -85,B 0,C 180,E1 4154.265,E2 4154.265} C_VEL
LIN {X 0,Y 111.444,Z 1175.074,A -85,B 0,C 180,E1 4141.542,E2 4141.542} C_VEL
LIN {X 0,Y 105.093,Z 1176.551,A -85,B 0,C 180,E1 4123.415,E2 4123.415} C_VEL
LIN {X 0,Y 113.551,Z 1177.599,A -85,B 0,C 180,E1 4102.429,E2 4102.429} C_VEL
LIN {X 0,Y 113.706,Z 1177.678,A -85,B 0,C 180,E1 4101.918,E2 4101.918} C_VEL
LIN {X 0,Y 99.821,Z 1182.485,A -85,B 0,C 180,E1 4089.137,E2 4089.137} C_VEL
LIN {X 0,Y 92.005,Z 1185.223,A -85,B 0,C 180,E1 4075.775,E2 4075.775} C_VEL
LIN {X 0,Y 88.62,Z 1186.733,A -85,B 0,C 180,E1 4061.726,E2 4061.726} C_VEL
LIN {X 0,Y 88.101,Z 1187.084,A -85,B 0,C 180,E1 4051.309,E2 4051.309} C_VEL
LIN {X 0,Y 88.321,Z 1186.884,A -85,B 0,C 180,E1 4041.545,E2 4041.545} C_VEL
LIN {X 0,Y 90.664,Z 1185.83,A -85,B 0,C 180,E1 4027.986,E2 4027.986} C_VEL
LIN {X 0,Y 97.308,Z 1183.334,A -85,B 0,C 180,E1 4014.157,E2 4014.157} C_VEL
LIN {X 0,Y 108.679,Z 1179.506,A -85,B 0,C 180,E1 4001.832,E2 4001.832} C_VEL
LIN {X 0,Y 124.565,Z 1173.775,A -85,B 0,C 180,E1 3991.45,E2 3991.45} C_VEL
LIN {X 0,Y 142.908,Z 1166.743,A -85,B 0,C 180,E1 3983.584,E2 3983.584} C_VEL
LIN {X 0,Y 163.449,Z 1157.792,A -85,B 0,C 180,E1 3977.402,E2 3977.402} C_VEL
LIN {X 0,Y 185.41,Z 1147.058,A -85,B 0,C 180,E1 3972.572,E2 3972.572} C_VEL
LIN {X 0,Y 206.511,Z 1135.562,A -85,B 0,C 180,E1 3969.011,E2 3969.011} C_VEL
LIN {X 0,Y 226.329,Z 1123.232,A -85,B 0,C 180,E1 3966.307,E2 3966.307} C_VEL
LIN {X 0,Y 245.595,Z 1110.187,A -85,B 0,C 180,E1 3964.131,E2 3964.131} C_VEL
LIN {X 0,Y 265.159,Z 1095.192,A -85,B 0,C 180,E1 3962.249,E2 3962.249} C_VEL
LIN {X 0,Y 284.693,Z 1078.529,A -85,B 0,C 180,E1 3960.611,E2 3960.611} C_VEL
LIN {X 0,Y 264.003,Z 1097.014,A -85,B 0,C 180,E1 3958.906,E2 3958.906} C_VEL
LIN {X 0,Y 246.251,Z 1111.222,A -85,B 0,C 180,E1 3957.197,E2 3957.197} C_VEL
LIN {X 0,Y 224.894,Z 1126.519,A -85,B 0,C 180,E1 3954.775,E2 3954.775} C_VEL
LIN {X 0,Y 216.98,Z 1131.824,A -85,B 0,C 180,E1 3953.743,E2 3953.743} C_VEL
LIN {X 0,Y 210.689,Z 1135.825,A -85,B 0,C 180,E1 3953.16,E2 3953.16} C_VEL
LIN {X 0,Y 192.157,Z 1145.868,A -85,B 0,C 180,E1 3952.383,E2 3952.383} C_VEL
LIN {X 0,Y 186.531,Z 1148.723,A -85,B 0,C 180,E1 3951.734,E2 3951.734} C_VEL
LIN {X 0,Y 165.716,Z 1159.177,A -85,B 0,C 180,E1 3947.79,E2 3947.79} C_VEL
LIN {X 0,Y 143.836,Z 1168.981,A -85,B 0,C 180,E1 3942.226,E2 3942.226} C_VEL
LIN {X 0,Y 123.629,Z 1176.952,A -85,B 0,C 180,E1 3934.92,E2 3934.92} C_VEL
LIN {X 0,Y 105.933,Z 1183.127,A -85,B 0,C 180,E1 3925.19,E2 3925.19} C_VEL
LIN {X 0,Y 91.949,Z 1187.814,A -85,B 0,C 180,E1 3912.382,E2 3912.382} C_VEL
LIN {X 0,Y 83.342,Z 1190.732,A -85,B 0,C 180,E1 3897.113,E2 3897.113} C_VEL
LIN {X 0,Y 80.23,Z 1192.307,A -85,B 0,C 180,E1 3881.493,E2 3881.493} C_VEL
LIN {X 0,Y 80.091,Z 1192.611,A -85,B 0,C 180,E1 3871.422,E2 3871.422} C_VEL
LIN {X 0,Y 80.101,Z 1192.424,A -85,B 0,C 180,E1 3862.099,E2 3862.099} C_VEL
LIN {X 0,Y 81.866,Z 1191.392,A -85,B 0,C 180,E1 3847.742,E2 3847.742} C_VEL
LIN {X 0,Y 89.321,Z 1188.63,A -85,B 0,C 180,E1 3831.17,E2 3831.17} C_VEL
LIN {X 0,Y 103.424,Z 1183.979,A -85,B 0,C 180,E1 3816.627,E2 3816.627} C_VEL
LIN {X 0,Y 121.373,Z 1177.735,A -85,B 0,C 180,E1 3806.098,E2 3806.098} C_VEL
LIN {X 0,Y 130.901,Z 1174.085,A -85,B 0,C 180,E1 3802.045,E2 3802.045} C_VEL
LIN {X 0,Y 112.824,Z 1176.131,A -85,B 0,C 180,E1 3791.761,E2 3791.761} C_VEL
LIN {X 0,Y 99.083,Z 1177.845,A -85,B 0,C 180,E1 3773.627,E2 3773.627} C_VEL
LIN {X 0,Y 99.576,Z 1178.899,A -85,B 0,C 180,E1 3751.839,E2 3751.839} C_VEL
LIN {X 0,Y 104.795,Z 1179.308,A -85,B 0,C 180,E1 3742.601,E2 3742.601} C_VEL
LIN {X 0,Y 91.261,Z 1183.462,A -85,B 0,C 180,E1 3729.464,E2 3729.464} C_VEL
LIN {X 0,Y 83.126,Z 1186.094,A -85,B 0,C 180,E1 3713.911,E2 3713.911} C_VEL
LIN {X 0,Y 80.382,Z 1187.145,A -85,B 0,C 180,E1 3699.315,E2 3699.315} C_VEL
LIN {X 0,Y 80.105,Z 1187.353,A -85,B 0,C 180,E1 3688.578,E2 3688.578} C_VEL
LIN {X 0,Y 80.721,Z 1187.019,A -85,B 0,C 180,E1 3677.126,E2 3677.126} C_VEL
LIN {X 0,Y 84.683,Z 1185.518,A -85,B 0,C 180,E1 3661.826,E2 3661.826} C_VEL
LIN {X 0,Y 93.034,Z 1182.949,A -85,B 0,C 180,E1 3648.225,E2 3648.225} C_VEL
LIN {X 0,Y 107.728,Z 1178.343,A -85,B 0,C 180,E1 3635.249,E2 3635.249} C_VEL
LIN {X 0,Y 124.705,Z 1172.664,A -85,B 0,C 180,E1 3626.116,E2 3626.116} C_VEL
LIN {X 0,Y 144.765,Z 1165.05,A -85,B 0,C 180,E1 3618.888,E2 3618.888} C_VEL
LIN {X 0,Y 166.492,Z 1155.807,A -85,B 0,C 180,E1 3613.389,E2 3613.389} C_VEL
LIN {X 0,Y 186.577,Z 1146.008,A -85,B 0,C 180,E1 3609.563,E2 3609.563} C_VEL
LIN {X 0,Y 207.278,Z 1134.844,A -85,B 0,C 180,E1 3606.461,E2 3606.461} C_VEL
LIN {X 0,Y 227.514,Z 1122.523,A -85,B 0,C 180,E1 3604.002,E2 3604.002} C_VEL
LIN {X 0,Y 249.084,Z 1107.769,A -85,B 0,C 180,E1 3601.834,E2 3601.834} C_VEL
LIN {X 0,Y 262.67,Z 1097.553,A -85,B 0,C 180,E1 3600.631,E2 3600.631} C_VEL
LIN {X 0,Y 242.012,Z 1113.738,A -85,B 0,C 180,E1 3598.786,E2 3598.786} C_VEL
LIN {X 0,Y 221.351,Z 1127.95,A -85,B 0,C 180,E1 3596.595,E2 3596.595} C_VEL
LIN {X 0,Y 200.117,Z 1141.126,A -85,B 0,C 180,E1 3593.843,E2 3593.843} C_VEL
LIN {X 0,Y 186.531,Z 1148.723,A -85,B 0,C 180,E1 3591.734,E2 3591.734} C_VEL
LIN {X 0,Y 179.919,Z 1151.984,A -85,B 0,C 180,E1 3590.958,E2 3590.958} C_VEL
LIN {X 0,Y 160.798,Z 1160.492,A -85,B 0,C 180,E1 3589.708,E2 3589.708} C_VEL
LIN {X 0,Y 155.111,Z 1162.865,A -85,B 0,C 180,E1 3588.808,E2 3588.808} C_VEL
LIN {X 0,Y 135.072,Z 1171.122,A -85,B 0,C 180,E1 3583.662,E2 3583.662} C_VEL
LIN {X 0,Y 113.955,Z 1178.753,A -85,B 0,C 180,E1 3575.842,E2 3575.842} C_VEL
LIN {X 0,Y 96.001,Z 1184.557,A -85,B 0,C 180,E1 3565.354,E2 3565.354} C_VEL
LIN {X 0,Y 81.834,Z 1188.698,A -85,B 0,C 180,E1 3550.751,E2 3550.751} C_VEL
LIN {X 0,Y 73.75,Z 1191.31,A -85,B 0,C 180,E1 3532.299,E2 3532.299} C_VEL
LIN {X 0,Y 72.105,Z 1192.181,A -85,B 0,C 180,E1 3517.961,E2 3517.961} C_VEL
LIN {X 0,Y 72.094,Z 1192.345,A -85,B 0,C 180,E1 3508.401,E2 3508.401} C_VEL
LIN {X 0,Y 72.31,Z 1192.03,A -85,B 0,C 180,E1 3497.208,E2 3497.208} C_VEL
LIN {X 0,Y 76.115,Z 1190.458,A -85,B 0,C 180,E1 3480.044,E2 3480.044} C_VEL
LIN {X 0,Y 86.53,Z 1187.348,A -85,B 0,C 180,E1 3463.271,E2 3463.271} C_VEL
LIN {X 0,Y 102.802,Z 1182.345,A -85,B 0,C 180,E1 3450.032,E2 3450.032} C_VEL
LIN {X 0,Y 119.329,Z 1176.91,A -85,B 0,C 180,E1 3441.823,E2 3441.823} C_VEL
LIN {X 0,Y 99.795,Z 1178.728,A -85,B 0,C 180,E1 3428.064,E2 3428.064} C_VEL
LIN {X 0,Y 89.919,Z 1179.932,A -85,B 0,C 180,E1 3408.144,E2 3408.144} C_VEL
LIN {X 0,Y 94.671,Z 1180.727,A -85,B 0,C 180,E1 3385.226,E2 3385.226} C_VEL
LIN {X 0,Y 95.709,Z 1180.802,A -85,B 0,C 180,E1 3383.294,E2 3383.294} C_VEL
LIN {X 0,Y 82.248,Z 1184.537,A -85,B 0,C 180,E1 3369.22,E2 3369.22} C_VEL
LIN {X 0,Y 74.354,Z 1186.729,A -85,B 0,C 180,E1 3351.89,E2 3351.89} C_VEL
LIN {X 0,Y 72.286,Z 1187.463,A -85,B 0,C 180,E1 3337.961,E2 3337.961} C_VEL
LIN {X 0,Y 72.114,Z 1187.595,A -85,B 0,C 180,E1 3327.626,E2 3327.626} C_VEL
LIN {X 0,Y 72.973,Z 1187.227,A -85,B 0,C 180,E1 3314.92,E2 3314.92} C_VEL
LIN {X 0,Y 77.571,Z 1185.79,A -85,B 0,C 180,E1 3298.973,E2 3298.973} C_VEL
LIN {X 0,Y 87.343,Z 1183.171,A -85,B 0,C 180,E1 3284.292,E2 3284.292} C_VEL
LIN {X 0,Y 103.162,Z 1178.662,A -85,B 0,C 180,E1 3271.482,E2 3271.482} C_VEL
LIN {X 0,Y 122.079,Z 1172.741,A -85,B 0,C 180,E1 3262.269,E2 3262.269} C_VEL
LIN {X 0,Y 142.284,Z 1165.388,A -85,B 0,C 180,E1 3255.708,E2 3255.708} C_VEL
LIN {X 0,Y 163.844,Z 1156.606,A -85,B 0,C 180,E1 3250.752,E2 3250.752} C_VEL
LIN {X 0,Y 185.358,Z 1146.451,A -85,B 0,C 180,E1 3247.03,E2 3247.03} C_VEL
LIN {X 0,Y 207.481,Z 1134.69,A -85,B 0,C 180,E1 3244.053,E2 3244.053} C_VEL
LIN {X 0,Y 228.074,Z 1122.418,A -85,B 0,C 180,E1 3241.823,E2 3241.823} C_VEL
LIN {X 0,Y 240.514,Z 1114.232,A -85,B 0,C 180,E1 3240.661,E2 3240.661} C_VEL
LIN {X 0,Y 220.018,Z 1128.136,A -85,B 0,C 180,E1 3238.682,E2 3238.682} C_VEL
LIN {X 0,Y 197.44,Z 1141.701,A -85,B 0,C 180,E1 3236.014,E2 3236.014} C_VEL
LIN {X 0,Y 178.221,Z 1151.958,A -85,B 0,C 180,E1 3233.194,E2 3233.194} C_VEL
LIN {X 0,Y 155.111,Z 1162.865,A -85,B 0,C 180,E1 3228.808,E2 3228.808} C_VEL
LIN {X 0,Y 148.422,Z 1165.616,A -85,B 0,C 180,E1 3227.713,E2 3227.713} C_VEL
LIN {X 0,Y 128.909,Z 1172.402,A -85,B 0,C 180,E1 3225.641,E2 3225.641} C_VEL
LIN {X 0,Y 123.231,Z 1174.24,A -85,B 0,C 180,E1 3224.317,E2 3224.317} C_VEL
LIN {X 0,Y 102.722,Z 1180.974,A -85,B 0,C 180,E1 3216.186,E2 3216.186} C_VEL
LIN {X 0,Y 84.745,Z 1186.038,A -85,B 0,C 180,E1 3204.484,E2 3204.484} C_VEL
LIN {X 0,Y 70.967,Z 1189.677,A -85,B 0,C 180,E1 3187.277,E2 3187.277} C_VEL
LIN {X 0,Y 65.276,Z 1191.345,A -85,B 0,C 180,E1 3170.617,E2 3170.617} C_VEL
LIN {X 0,Y 64.08,Z 1191.981,A -85,B 0,C 180,E1 3156.26,E2 3156.26} C_VEL
LIN {X 0,Y 64.081,Z 1192.056,A -85,B 0,C 180,E1 3147.004,E2 3147.004} C_VEL
LIN {X 0,Y 64.639,Z 1191.628,A -85,B 0,C 180,E1 3133.55,E2 3133.55} C_VEL
LIN {X 0,Y 69.818,Z 1189.971,A -85,B 0,C 180,E1 3115.039,E2 3115.039} C_VEL
LIN {X 0,Y 82.253,Z 1186.718,A -85,B 0,C 180,E1 3097.787,E2 3097.787} C_VEL
LIN {X 0,Y 99.636,Z 1181.807,A -85,B 0,C 180,E1 3085.405,E2 3085.405} C_VEL
LIN {X 0,Y 107.646,Z 1179.338,A -85,B 0,C 180,E1 3081.388,E2 3081.388} C_VEL
LIN {X 0,Y 90.164,Z 1180.711,A -85,B 0,C 180,E1 3067.007,E2 3067.007} C_VEL
LIN {X 0,Y 81.695,Z 1181.734,A -85,B 0,C 180,E1 3044.379,E2 3044.379} C_VEL
LIN {X 0,Y 86.671,Z 1182.204,A -85,B 0,C 180,E1 3024.168,E2 3024.168} C_VEL
LIN {X 0,Y 72.341,Z 1185.677,A -85,B 0,C 180,E1 3007.468,E2 3007.468} C_VEL
LIN {X 0,Y 65.865,Z 1187.257,A -85,B 0,C 180,E1 2990.447,E2 2990.447} C_VEL
LIN {X 0,Y 64.203,Z 1187.78,A -85,B 0,C 180,E1 2976.27,E2 2976.27} C_VEL
LIN {X 0,Y 64.146,Z 1187.819,A -85,B 0,C 180,E1 2965.541,E2 2965.541} C_VEL
LIN {X 0,Y 65.544,Z 1187.362,A -85,B 0,C 180,E1 2951.055,E2 2951.055} C_VEL
LIN {X 0,Y 71.193,Z 1185.95,A -85,B 0,C 180,E1 2934.548,E2 2934.548} C_VEL
LIN {X 0,Y 83.894,Z 1183.001,A -85,B 0,C 180,E1 2918.144,E2 2918.144} C_VEL
LIN {X 0,Y 101.357,Z 1178.336,A -85,B 0,C 180,E1 2906.158,E2 2906.158} C_VEL
LIN {X 0,Y 122.583,Z 1171.927,A -85,B 0,C 180,E1 2897.401,E2 2897.401} C_VEL
LIN {X 0,Y 143.901,Z 1164.405,A -85,B 0,C 180,E1 2891.584,E2 2891.584} C_VEL
LIN {X 0,Y 166.279,Z 1155.261,A -85,B 0,C 180,E1 2887.204,E2 2887.204} C_VEL
LIN {X 0,Y 188.413,Z 1145.056,A -85,B 0,C 180,E1 2883.956,E2 2883.956} C_VEL
LIN {X 0,Y 212.012,Z 1132.397,A -85,B 0,C 180,E1 2881.251,E2 2881.251} C_VEL
LIN {X 0,Y 217.802,Z 1129.072,A -85,B 0,C 180,E1 2880.679,E2 2880.679} C_VEL
LIN {X 0,Y 196.044,Z 1141.811,A -85,B 0,C 180,E1 2878.356,E2 2878.356} C_VEL
LIN {X 0,Y 174.508,Z 1153.035,A -85,B 0,C 180,E1 2875.481,E2 2875.481} C_VEL
LIN {X 0,Y 152.572,Z 1162.921,A -85,B 0,C 180,E1 2871.687,E2 2871.687} C_VEL
LIN {X 0,Y 131.795,Z 1171.225,A -85,B 0,C 180,E1 2866.844,E2 2866.844} C_VEL
LIN {X 0,Y 123.231,Z 1174.24,A -85,B 0,C 180,E1 2864.317,E2 2864.317} C_VEL
LIN {X 0,Y 116.605,Z 1176.444,A -85,B 0,C 180,E1 2862.664,E2 2862.664} C_VEL
LIN {X 0,Y 97.149,Z 1181.426,A -85,B 0,C 180,E1 2858.924,E2 2858.924} C_VEL
LIN {X 0,Y 91.693,Z 1182.783,A -85,B 0,C 180,E1 2856.76,E2 2856.76} C_VEL
LIN {X 0,Y 72.85,Z 1187.49,A -85,B 0,C 180,E1 2842.739,E2 2842.739} C_VEL
LIN {X 0,Y 61.201,Z 1190.212,A -85,B 0,C 180,E1 2824.863,E2 2824.863} C_VEL
LIN {X 0,Y 56.321,Z 1191.578,A -85,B 0,C 180,E1 2803.331,E2 2803.331} C_VEL
LIN {X 0,Y 56.103,Z 1191.843,A -85,B 0,C 180,E1 2791.009,E2 2791.009} C_VEL
LIN {X 0,Y 56.206,Z 1191.623,A -85,B 0,C 180,E1 2778.703,E2 2778.703} C_VEL
LIN {X 0,Y 60.159,Z 1190.49,A -85,B 0,C 180,E1 2757.855,E2 2757.855} C_VEL
LIN {X 0,Y 71.637,Z 1187.74,A -85,B 0,C 180,E1 2738.575,E2 2738.575} C_VEL
LIN {X 0,Y 89.916,Z 1183.25,A -85,B 0,C 180,E1 2724.219,E2 2724.219} C_VEL
LIN {X 0,Y 96.162,Z 1181.537,A -85,B 0,C 180,E1 2720.919,E2 2720.919} C_VEL
LIN {X 0,Y 78.481,Z 1182.696,A -85,B 0,C 180,E1 2702.19,E2 2702.19} C_VEL
LIN {X 0,Y 75.499,Z 1183.434,A -85,B 0,C 180,E1 2671.525,E2 2671.525} C_VEL
LIN {X 0,Y 77.762,Z 1183.517,A -85,B 0,C 180,E1 2665.394,E2 2665.394} C_VEL
LIN {X 0,Y 64.146,Z 1186.321,A -85,B 0,C 180,E1 2648.586,E2 2648.586} C_VEL
LIN {X 0,Y 57.349,Z 1187.797,A -85,B 0,C 180,E1 2628.303,E2 2628.303} C_VEL
LIN {X 0,Y 56.128,Z 1188.115,A -85,B 0,C 180,E1 2613.076,E2 2613.076} C_VEL
LIN {X 0,Y 56.341,Z 1188.014,A -85,B 0,C 180,E1 2600.822,E2 2600.822} C_VEL
LIN {X 0,Y 59.119,Z 1187.367,A -85,B 0,C 180,E1 2583.69,E2 2583.69} C_VEL
LIN {X 0,Y 69.105,Z 1185.409,A -85,B 0,C 180,E1 2563.675,E2 2563.675} C_VEL
LIN {X 0,Y 85.594,Z 1181.714,A -85,B 0,C 180,E1 2548.617,E2 2548.617} C_VEL
LIN {X 0,Y 106.335,Z 1176.409,A -85,B 0,C 180,E1 2538.27,E2 2538.27} C_VEL
LIN {X 0,Y 127.603,Z 1169.921,A -85,B 0,C 180,E1 2531.656,E2 2531.656} C_VEL
LIN {X 0,Y 150.039,Z 1161.891,A -85,B 0,C 180,E1 2526.846,E2 2526.846} C_VEL
LIN {X 0,Y 172.755,Z 1152.574,A -85,B 0,C 180,E1 2523.318,E2 2523.318} C_VEL
LIN {X 0,Y 194.662,Z 1142.097,A -85,B 0,C 180,E1 2520.694,E2 2520.694} C_VEL
LIN {X 0,Y 171.085,Z 1154.012,A -85,B 0,C 180,E1 2517.867,E2 2517.867} C_VEL
LIN {X 0,Y 149.654,Z 1163.338,A -85,B 0,C 180,E1 2514.514,E2 2514.514} C_VEL
LIN {X 0,Y 127.018,Z 1171.971,A -85,B 0,C 180,E1 2509.702,E2 2509.702} C_VEL
LIN {X 0,Y 106.427,Z 1178.586,A -85,B 0,C 180,E1 2503.37,E2 2503.37} C_VEL
LIN {X 0,Y 91.693,Z 1182.783,A -85,B 0,C 180,E1 2496.76,E2 2496.76} C_VEL
LIN {X 0,Y 85.41,Z 1184.307,A -85,B 0,C 180,E1 2493.97,E2 2493.97} C_VEL
LIN {X 0,Y 66.57,Z 1187.618,A -85,B 0,C 180,E1 2485.968,E2 2485.968} C_VEL
LIN {X 0,Y 62.322,Z 1188.439,A -85,B 0,C 180,E1 2482.117,E2 2482.117} C_VEL
LIN {X 0,Y 50.891,Z 1190.681,A -85,B 0,C 180,E1 2459.403,E2 2459.403} C_VEL
LIN {X 0,Y 48.118,Z 1191.453,A -85,B 0,C 180,E1 2438.349,E2 2438.349} C_VEL
LIN {X 0,Y 48.091,Z 1191.556,A -85,B 0,C 180,E1 2427.602,E2 2427.602} C_VEL
LIN {X 0,Y 48.849,Z 1191.226,A -85,B 0,C 180,E1 2410.868,E2 2410.868} C_VEL
LIN {X 0,Y 56.519,Z 1189.519,A -85,B 0,C 180,E1 2386.498,E2 2386.498} C_VEL
LIN {X 0,Y 71.741,Z 1186.455,A -85,B 0,C 180,E1 2368.572,E2 2368.572} C_VEL
LIN {X 0,Y 84.682,Z 1183.491,A -85,B 0,C 180,E1 2360.223,E2 2360.223} C_VEL
